LIN {X 89.055,Y 275.987,Z 202.901,A -107.884,B 90.000,C 0.000} C_DIS
LIN {X 91.283,Y 275.258,Z 203.769,A -108.347,B 90.000,C 0.000} C_DIS
LIN {X 93.519,Y 274.506,Z 204.596,A -108.813,B 90.000,C 0.000} C_DIS
LIN {X 95.762,Y 273.732,Z 205.382,A -109.282,B 90.000,C 0.000} C_DIS
LIN {X 98.010,Y 272.935,Z 206.132,A -109.753,B 90.000,C 0.000} C_DIS
LIN {X 100.260,Y 272.116,Z 206.848,A -110.226,B 90.000,C 0.000} C_DIS
LIN {X 102.512,Y 271.277,Z 207.537,A -110.701,B 90.000,C 0.000} C_DIS
LIN {X 104.763,Y 270.415,Z 208.199,A -111.177,B 90.000,C 0.000} C_DIS
LIN {X 107.012,Y 269.533,Z 208.839,A -111.655,B 90.000,C 0.000} C_DIS
LIN {X 109.259,Y 268.630,Z 209.461,A -112.133,B 90.000,C 0.000} C_DIS
LIN {X 111.501,Y 267.707,Z 210.069,A -112.612,B 90.000,C 0.000} C_DIS
LIN {X 113.738,Y 266.764,Z 210.665,A -113.092,B 90.000,C 0.000} C_DIS
LIN {X 115.968,Y 265.800,Z 211.254,A -113.571,B 90.000,C 0.000} C_DIS
LIN {X 118.189,Y 264.816,Z 211.841,A -114.052,B 90.000,C 0.000} C_DIS
LIN {X 120.405,Y 263.818,Z 212.427,A -114.532,B 90.000,C 0.000} C_DIS
LIN {X 122.611,Y 262.801,Z 213.018,A -115.012,B 90.000,C 0.000} C_DIS
LIN {X 124.806,Y 261.767,Z 213.616,A -115.491,B 90.000,C 0.000} C_DIS
LIN {X 126.991,Y 260.715,Z 214.224,A -115.970,B 90.000,C 0.000} C_DIS
LIN {X 129.163,Y 259.646,Z 214.847,A -116.448,B 90.000,C 0.000} C_DIS
LIN {X 131.322,Y 258.561,Z 215.489,A -116.926,B 90.000,C 0.000} C_DIS
LIN {X 133.467,Y 257.462,Z 216.152,A -117.402,B 90.000,C 0.000} C_DIS
LIN {X 135.595,Y 256.346,Z 216.842,A -117.877,B 90.000,C 0.000} C_DIS
LIN {X 137.706,Y 255.218,Z 217.561,A -118.350,B 90.000,C 0.000} C_DIS
LIN {X 139.800,Y 254.078,Z 218.313,A -118.821,B 90.000,C 0.000} C_DIS
LIN {X 141.874,Y 252.926,Z 219.100,A -119.289,B 90.000,C 0.000} C_DIS
LIN {X 143.243,Y 252.153,Z 219.646,A -119.600,B 90.000,C 0.000} C_DIS
LIN {X 142.255,Y 250.414,Z 219.646,A -119.600,B 90.000,C 0.000} C_DIS
WAIT SEC 0.1
RET=EKI_SetBool("oxy","torchState",FALSE)
RET = EKI_Send("oxy","torchState")
LIN {X 133.364,Y 234.764,Z 219.646,A -119.600,B 90.000,C 0.000} C_DIS
LIN {X 126.224,Y 238.679,Z 194.850,A -117.872,B 90.000,C 0.000} C_DIS
LIN {X 134.638,Y 254.591,Z 194.850,A -117.872,B 90.000,C 0.000} C_DIS
LIN {X 135.573,Y 256.359,Z 194.850,A -117.872,B 90.000,C 0.000} C_DIS
WAIT SEC 1.75
RET=EKI_SetBool("oxy","torchState",TRUE)
RET = EKI_Send("oxy","torchState")
LIN {X 137.702,Y 255.221,Z 195.499,A -118.349,B 90.000,C 0.000} C_DIS
LIN {X 139.833,Y 254.060,Z 196.100,A -118.828,B 90.000,C 0.000} C_DIS
LIN {X 141.962,Y 252.876,Z 196.661,A -119.309,B 90.000,C 0.000} C_DIS
LIN {X 144.088,Y 251.672,Z 197.189,A -119.792,B 90.000,C 0.000} C_DIS
LIN {X 146.208,Y 250.445,Z 197.689,A -120.276,B 90.000,C 0.000} C_DIS
LIN {X 148.321,Y 249.199,Z 198.169,A -120.761,B 90.000,C 0.000} C_DIS
LIN {X 150.425,Y 247.933,Z 198.638,A -121.246,B 90.000,C 0.000} C_DIS
LIN {X 152.518,Y 246.648,Z 199.103,A -121.731,B 90.000,C 0.000} C_DIS
LIN {X 154.603,Y 245.350,Z 199.569,A -122.216,B 90.000,C 0.000} C_DIS
LIN {X 156.674,Y 244.034,Z 200.044,A -122.701,B 90.000,C 0.000} C_DIS
LIN {X 158.730,Y 242.701,Z 200.536,A -123.185,B 90.000,C 0.000} C_DIS
LIN {X 159.559,Y 242.159,Z 200.740,A -123.381,B 90.000,C 0.000} C_DIS
LIN {X 158.459,Y 240.488,Z 200.740,A -123.381,B 90.000,C 0.000} C_DIS
WAIT SEC 0.1
RET=EKI_SetBool("oxy","torchState",FALSE)
RET = EKI_Send("oxy","torchState")
LIN {X 148.555,Y 225.458,Z 200.740,A -123.381,B 90.000,C 0.000} C_DIS
LIN {X 166.339,Y 212.677,Z 183.902,A -128.030,B 90.000,C 0.000} C_DIS
LIN {X 177.428,Y 226.855,Z 183.902,A -128.030,B 90.000,C 0.000} C_DIS
LIN {X 178.660,Y 228.430,Z 183.902,A -128.030,B 90.000,C 0.000} C_DIS
WAIT SEC 1.75
RET=EKI_SetBool("oxy","torchState",TRUE)
RET = EKI_Send("oxy","torchState")
LIN {X 180.589,Y 226.908,Z 184.361,A -128.515,B 90.000,C 0.000} C_DIS
LIN {X 182.507,Y 225.367,Z 184.805,A -129.001,B 90.000,C 0.000} C_DIS
LIN {X 184.414,Y 223.810,Z 185.234,A -129.488,B 90.000,C 0.000} C_DIS
LIN {X 186.310,Y 222.234,Z 185.649,A -129.975,B 90.000,C 0.000} C_DIS
LIN {X 188.194,Y 220.640,Z 186.048,A -130.462,B 90.000,C 0.000} C_DIS
LIN {X 190.067,Y 219.029,Z 186.431,A -130.950,B 90.000,C 0.000} C_DIS
LIN {X 191.927,Y 217.401,Z 186.799,A -131.439,B 90.000,C 0.000} C_DIS
LIN {X 193.776,Y 215.755,Z 187.150,A -131.928,B 90.000,C 0.000} C_DIS
LIN {X 195.612,Y 214.092,Z 187.486,A -132.417,B 90.000,C 0.000} C_DIS
LIN {X 197.435,Y 212.412,Z 187.804,A -132.907,B 90.000,C 0.000} C_DIS
LIN {X 199.245,Y 210.715,Z 188.106,A -133.397,B 90.000,C 0.000} C_DIS
LIN {X 201.043,Y 209.002,Z 188.392,A -133.888,B 90.000,C 0.000} C_DIS
LIN {X 202.826,Y 207.271,Z 188.659,A -134.379,B 90.000,C 0.000} C_DIS
LIN {X 204.596,Y 205.524,Z 188.909,A -134.870,B 90.000,C 0.000} C_DIS
LIN {X 206.352,Y 203.760,Z 189.141,A -135.362,B 90.000,C 0.000} C_DIS
LIN {X 208.094,Y 201.980,Z 189.356,A -135.854,B 90.000,C 0.000} C_DIS
LIN {X 209.822,Y 200.184,Z 189.552,A -136.347,B 90.000,C 0.000} C_DIS
LIN {X 211.535,Y 198.372,Z 189.731,A -136.839,B 90.000,C 0.000} C_DIS
LIN {X 213.234,Y 196.545,Z 189.891,A -137.332,B 90.000,C 0.000} C_DIS
LIN {X 214.917,Y 194.703,Z 190.032,A -137.825,B 90.000,C 0.000} C_DIS
LIN {X 216.586,Y 192.846,Z 190.155,A -138.318,B 90.000,C 0.000} C_DIS
LIN {X 218.239,Y 190.973,Z 190.258,A -138.812,B 90.000,C 0.000} C_DIS
LIN {X 219.876,Y 189.087,Z 190.343,A -139.306,B 90.000,C 0.000} C_DIS
LIN {X 221.498,Y 187.185,Z 190.408,A -139.799,B 90.000,C 0.000} C_DIS
LIN {X 223.103,Y 185.270,Z 190.454,A -140.293,B 90.000,C 0.000} C_DIS
LIN {X 224.481,Y 183.598,Z 190.477,A -140.721,B 90.000,C 0.000} C_DIS
LIN {X 222.933,Y 182.331,Z 190.477,A -140.721,B 90.000,C 0.000} C_DIS
WAIT SEC 0.1
RET=EKI_SetBool("oxy","torchState",FALSE)
RET = EKI_Send("oxy","torchState")
LIN {X 209.000,Y 170.936,Z 190.477,A -140.721,B 90.000,C 0.000} C_DIS
LIN {X 223.386,Y 151.653,Z 212.037,A -145.828,B 90.000,C 0.000} C_DIS
LIN {X 238.278,Y 161.763,Z 212.037,A -145.828,B 90.000,C 0.000} C_DIS
LIN {X 239.933,Y 162.887,Z 212.037,A -145.828,B 90.000,C 0.000} C_DIS
WAIT SEC 1.75
RET=EKI_SetBool("oxy","torchState",TRUE)
RET = EKI_Send("oxy","torchState")
LIN {X 238.516,Y 164.946,Z 212.053,A -145.334,B 90.000,C 0.000} C_DIS
LIN {X 237.085,Y 166.995,Z 212.070,A -144.840,B 90.000,C 0.000} C_DIS
LIN {X 235.641,Y 169.035,Z 212.086,A -144.346,B 90.000,C 0.000} C_DIS
LIN {X 234.172,Y 171.058,Z 212.108,A -143.853,B 90.000,C 0.000} C_DIS
LIN {X 232.688,Y 173.069,Z 212.129,A -143.359,B 90.000,C 0.000} C_DIS
LIN {X 231.191,Y 175.071,Z 212.152,A -142.865,B 90.000,C 0.000} C_DIS
LIN {X 229.671,Y 177.055,Z 212.179,A -142.371,B 90.000,C 0.000} C_DIS
LIN {X 228.135,Y 179.028,Z 212.206,A -141.877,B 90.000,C 0.000} C_DIS
LIN {X 226.587,Y 180.990,Z 212.234,A -141.383,B 90.000,C 0.000} C_DIS
LIN {X 225.017,Y 182.935,Z 212.266,A -140.890,B 90.000,C 0.000} C_DIS
LIN {X 223.430,Y 184.866,Z 212.299,A -140.396,B 90.000,C 0.000} C_DIS
LIN {X 221.831,Y 186.787,Z 212.332,A -139.902,B 90.000,C 0.000} C_DIS
LIN {X 220.212,Y 188.691,Z 212.370,A -139.408,B 90.000,C 0.000} C_DIS
LIN {X 218.576,Y 190.581,Z 212.408,A -138.914,B 90.000,C 0.000} C_DIS
LIN {X 216.927,Y 192.459,Z 212.448,A -138.420,B 90.000,C 0.000} C_DIS
LIN {X 215.261,Y 194.322,Z 212.491,A -137.927,B 90.000,C 0.000} C_DIS
LIN {X 213.576,Y 196.168,Z 212.534,A -137.433,B 90.000,C 0.000} C_DIS
LIN {X 211.879,Y 198.003,Z 212.580,A -136.939,B 90.000,C 0.000} C_DIS
LIN {X 210.166,Y 199.822,Z 212.628,A -136.445,B 90.000,C 0.000} C_DIS
LIN {X 208.434,Y 201.624,Z 212.677,A -135.951,B 90.000,C 0.000} C_DIS
LIN {X 206.689,Y 203.414,Z 212.728,A -135.458,B 90.000,C 0.000} C_DIS
LIN {X 204.930,Y 205.189,Z 212.782,A -134.964,B 90.000,C 0.000} C_DIS
LIN {X 203.152,Y 206.945,Z 212.836,A -134.470,B 90.000,C 0.000} C_DIS
LIN {X 201.362,Y 208.688,Z 212.893,A -133.976,B 90.000,C 0.000} C_DIS
LIN {X 199.558,Y 210.418,Z 212.952,A -133.483,B 90.000,C 0.000} C_DIS
LIN {X 197.735,Y 212.127,Z 213.012,A -132.989,B 90.000,C 0.000} C_DIS
LIN {X 195.900,Y 213.824,Z 213.074,A -132.495,B 90.000,C 0.000} C_DIS
LIN {X 194.053,Y 215.506,Z 213.139,A -132.001,B 90.000,C 0.000} C_DIS
LIN {X 192.187,Y 217.169,Z 213.204,A -131.508,B 90.000,C 0.000} C_DIS
LIN {X 191.631,Y 217.664,Z 213.223,A -131.361,B 90.000,C 0.000} C_DIS
LIN {X 190.309,Y 216.163,Z 213.223,A -131.361,B 90.000,C 0.000} C_DIS
WAIT SEC 0.1
RET=EKI_SetBool("oxy","torchState",FALSE)
RET = EKI_Send("oxy","torchState")
LIN {X 178.415,Y 202.653,Z 213.223,A -131.361,B 90.000,C 0.000} C_DIS
LIN {X 175.571,Y 205.122,Z 236.485,A -130.561,B 90.000,C 0.000} C_DIS
LIN {X 187.276,Y 218.796,Z 236.485,A -130.561,B 90.000,C 0.000} C_DIS
LIN {X 188.576,Y 220.316,Z 236.485,A -130.561,B 90.000,C 0.000} C_DIS
WAIT SEC 1.75
RET=EKI_SetBool("oxy","torchState",TRUE)
RET = EKI_Send("oxy","torchState")
LIN {X 190.445,Y 218.694,Z 236.131,A -131.050,B 90.000,C 0.000} C_DIS
LIN {X 192.308,Y 217.065,Z 235.780,A -131.539,B 90.000,C 0.000} C_DIS
LIN {X 194.151,Y 215.411,Z 235.439,A -132.029,B 90.000,C 0.000} C_DIS
LIN {X 195.984,Y 213.745,Z 235.101,A -132.518,B 90.000,C 0.000} C_DIS
LIN {X 197.805,Y 212.065,Z 234.769,A -133.007,B 90.000,C 0.000} C_DIS
LIN {X 199.608,Y 210.363,Z 234.446,A -133.497,B 90.000,C 0.000} C_DIS
LIN {X 201.401,Y 208.652,Z 234.126,A -133.987,B 90.000,C 0.000} C_DIS
LIN {X 203.177,Y 206.921,Z 233.814,A -134.477,B 90.000,C 0.000} C_DIS
LIN {X 204.939,Y 205.174,Z 233.507,A -134.967,B 90.000,C 0.000} C_DIS
LIN {X 206.691,Y 203.417,Z 233.205,A -135.457,B 90.000,C 0.000} C_DIS
LIN {X 208.420,Y 201.636,Z 232.913,A -135.948,B 90.000,C 0.000} C_DIS
LIN {X 210.140,Y 199.845,Z 232.624,A -136.438,B 90.000,C 0.000} C_DIS
LIN {X 211.845,Y 198.039,Z 232.341,A -136.929,B 90.000,C 0.000} C_DIS
LIN {X 213.532,Y 196.215,Z 232.066,A -137.420,B 90.000,C 0.000} C_DIS
LIN {X 215.209,Y 194.381,Z 231.795,A -137.911,B 90.000,C 0.000} C_DIS
LIN {X 216.864,Y 192.527,Z 231.532,A -138.402,B 90.000,C 0.000} C_DIS
LIN {X 218.507,Y 190.660,Z 231.274,A -138.893,B 90.000,C 0.000} C_DIS
LIN {X 220.137,Y 188.782,Z 231.021,A -139.385,B 90.000,C 0.000} C_DIS
LIN {X 221.745,Y 186.883,Z 230.777,A -139.876,B 90.000,C 0.000} C_DIS
LIN {X 223.342,Y 184.976,Z 230.537,A -140.368,B 90.000,C 0.000} C_DIS
LIN {X 224.921,Y 183.052,Z 230.304,A -140.860,B 90.000,C 0.000} C_DIS
LIN {X 226.482,Y 181.113,Z 230.077,A -141.351,B 90.000,C 0.000} C_DIS
LIN {X 228.033,Y 179.165,Z 229.855,A -141.843,B 90.000,C 0.000} C_DIS
LIN {X 229.559,Y 177.197,Z 229.641,A -142.335,B 90.000,C 0.000} C_DIS
LIN {X 231.074,Y 175.219,Z 229.432,A -142.828,B 90.000,C 0.000} C_DIS
LIN {X 232.573,Y 173.229,Z 229.229,A -143.320,B 90.000,C 0.000} C_DIS
LIN {X 234.049,Y 171.222,Z 229.033,A -143.812,B 90.000,C 0.000} C_DIS
LIN {X 235.515,Y 169.206,Z 228.842,A -144.305,B 90.000,C 0.000} C_DIS
LIN {X 236.960,Y 167.174,Z 228.658,A -144.797,B 90.000,C 0.000} C_DIS
LIN {X 238.387,Y 165.130,Z 228.480,A -145.290,B 90.000,C 0.000} C_DIS
LIN {X 239.804,Y 163.077,Z 228.306,A -145.782,B 90.000,C 0.000} C_DIS
LIN {X 241.192,Y 161.005,Z 228.142,A -146.275,B 90.000,C 0.000} C_DIS
LIN {X 242.569,Y 158.925,Z 227.982,A -146.768,B 90.000,C 0.000} C_DIS
LIN {X 243.929,Y 156.834,Z 227.828,A -147.261,B 90.000,C 0.000} C_DIS
LIN {X 245.266,Y 154.727,Z 227.681,A -147.754,B 90.000,C 0.000} C_DIS
LIN {X 246.593,Y 152.613,Z 227.539,A -148.247,B 90.000,C 0.000} C_DIS
LIN {X 247.894,Y 150.483,Z 227.404,A -148.740,B 90.000,C 0.000} C_DIS
LIN {X 249.180,Y 148.343,Z 227.275,A -149.234,B 90.000,C 0.000} C_DIS
LIN {X 250.452,Y 146.195,Z 227.151,A -149.727,B 90.000,C 0.000} C_DIS
LIN {X 251.697,Y 144.030,Z 227.036,A -150.220,B 90.000,C 0.000} C_DIS
LIN {X 252.930,Y 141.859,Z 226.924,A -150.714,B 90.000,C 0.000} C_DIS
LIN {X 254.143,Y 139.675,Z 226.820,A -151.207,B 90.000,C 0.000} C_DIS
LIN {X 255.334,Y 137.480,Z 226.722,A -151.701,B 90.000,C 0.000} C_DIS
LIN {X 256.513,Y 135.278,Z 226.628,A -152.194,B 90.000,C 0.000} C_DIS
LIN {X 257.665,Y 133.061,Z 226.544,A -152.688,B 90.000,C 0.000} C_DIS
LIN {X 258.260,Y 131.917,Z 226.500,A -152.942,B 90.000,C 0.000} C_DIS
LIN {X 256.478,Y 131.007,Z 226.500,A -152.942,B 90.000,C 0.000} C_DIS
WAIT SEC 0.1
RET=EKI_SetBool("oxy","torchState",FALSE)
RET = EKI_Send("oxy","torchState")
LIN {X 240.449,Y 122.819,Z 226.500,A -152.942,B 90.000,C 0.000} C_DIS
LIN {X 242.380,Y 118.962,Z 209.835,A -153.858,B 90.000,C 0.000} C_DIS
LIN {X 258.538,Y 126.893,Z 209.835,A -153.858,B 90.000,C 0.000} C_DIS
LIN {X 260.334,Y 127.774,Z 209.835,A -153.858,B 90.000,C 0.000} C_DIS
WAIT SEC 1.75
RET=EKI_SetBool("oxy","torchState",TRUE)
RET = EKI_Send("oxy","torchState")
LIN {X 261.410,Y 125.557,Z 209.418,A -154.345,B 90.000,C 0.000} C_DIS
LIN {X 262.464,Y 123.338,Z 208.956,A -154.830,B 90.000,C 0.000} C_DIS
LIN {X 263.495,Y 121.118,Z 208.449,A -155.314,B 90.000,C 0.000} C_DIS
LIN {X 264.505,Y 118.898,Z 207.901,A -155.795,B 90.000,C 0.000} C_DIS
LIN {X 265.491,Y 116.679,Z 207.309,A -156.275,B 90.000,C 0.000} C_DIS
LIN {X 266.455,Y 114.460,Z 206.680,A -156.753,B 90.000,C 0.000} C_DIS
LIN {X 267.397,Y 112.243,Z 206.013,A -157.229,B 90.000,C 0.000} C_DIS
LIN {X 268.316,Y 110.027,Z 205.310,A -157.703,B 90.000,C 0.000} C_DIS
LIN {X 269.213,Y 107.813,Z 204.573,A -158.175,B 90.000,C 0.000} C_DIS
LIN {X 270.089,Y 105.601,Z 203.805,A -158.645,B 90.000,C 0.000} C_DIS
LIN {X 270.942,Y 103.392,Z 203.004,A -159.113,B 90.000,C 0.000} C_DIS
LIN {X 271.774,Y 101.185,Z 202.177,A -159.579,B 90.000,C 0.000} C_DIS
LIN {X 272.584,Y 98.981,Z 201.321,A -160.043,B 90.000,C 0.000} C_DIS
LIN {X 273.373,Y 96.779,Z 200.440,A -160.505,B 90.000,C 0.000} C_DIS
LIN {X 274.142,Y 94.579,Z 199.535,A -160.966,B 90.000,C 0.000} C_DIS
LIN {X 274.891,Y 92.381,Z 198.609,A -161.424,B 90.000,C 0.000} C_DIS
LIN {X 275.620,Y 90.186,Z 197.661,A -161.881,B 90.000,C 0.000} C_DIS
LIN {X 276.327,Y 87.993,Z 196.693,A -162.337,B 90.000,C 0.000} C_DIS
LIN {X 277.015,Y 85.801,Z 195.707,A -162.790,B 90.000,C 0.000} C_DIS
LIN {X 277.684,Y 83.610,Z 194.706,A -163.243,B 90.000,C 0.000} C_DIS
LIN {X 278.219,Y 81.819,Z 193.877,A -163.612,B 90.000,C 0.000} C_DIS
LIN {X 276.300,Y 81.255,Z 193.877,A -163.612,B 90.000,C 0.000} C_DIS
WAIT SEC 0.1
RET=EKI_SetBool("oxy","torchState",FALSE)
RET = EKI_Send("oxy","torchState")
LIN {X 259.031,Y 76.177,Z 193.877,A -163.612,B 90.000,C 0.000} C_DIS
LIN {X 263.643,Y 58.244,Z 184.719,A -167.542,B 90.000,C 0.000} C_DIS
LIN {X 281.219,Y 62.127,Z 184.719,A -167.542,B 90.000,C 0.000} C_DIS
LIN {X 283.172,Y 62.558,Z 184.719,A -167.542,B 90.000,C 0.000} C_DIS
WAIT SEC 1.75
RET=EKI_SetBool("oxy","torchState",TRUE)
RET = EKI_Send("oxy","torchState")
LIN {X 283.654,Y 60.332,Z 183.689,A -167.992,B 90.000,C 0.000} C_DIS
LIN {X 284.118,Y 58.098,Z 182.669,A -168.443,B 90.000,C 0.000} C_DIS
LIN {X 284.566,Y 55.856,Z 181.657,A -168.895,B 90.000,C 0.000} C_DIS
LIN {X 284.999,Y 53.608,Z 180.653,A -169.347,B 90.000,C 0.000} C_DIS
LIN {X 285.416,Y 51.354,Z 179.657,A -169.800,B 90.000,C 0.000} C_DIS
LIN {X 285.810,Y 49.091,Z 178.670,A -170.254,B 90.000,C 0.000} C_DIS
LIN {X 286.190,Y 46.824,Z 177.689,A -170.708,B 90.000,C 0.000} C_DIS
LIN {X 286.556,Y 44.552,Z 176.713,A -171.163,B 90.000,C 0.000} C_DIS
LIN {X 286.896,Y 42.272,Z 175.746,A -171.618,B 90.000,C 0.000} C_DIS
LIN {X 287.229,Y 39.990,Z 174.781,A -172.074,B 90.000,C 0.000} C_DIS
LIN {X 287.537,Y 37.702,Z 173.823,A -172.530,B 90.000,C 0.000} C_DIS
LIN {X 287.826,Y 35.409,Z 172.870,A -172.987,B 90.000,C 0.000} C_DIS
LIN {X 288.096,Y 33.113,Z 171.920,A -173.443,B 90.000,C 0.000} C_DIS
LIN {X 288.355,Y 30.814,Z 170.973,A -173.900,B 90.000,C 0.000} C_DIS
LIN {X 288.593,Y 28.512,Z 170.029,A -174.358,B 90.000,C 0.000} C_DIS
LIN {X 288.809,Y 26.206,Z 169.087,A -174.815,B 90.000,C 0.000} C_DIS
LIN {X 289.006,Y 23.898,Z 168.148,A -175.273,B 90.000,C 0.000} C_DIS
LIN {X 289.188,Y 21.589,Z 167.209,A -175.731,B 90.000,C 0.000} C_DIS
LIN {X 289.351,Y 19.277,Z 166.271,A -176.188,B 90.000,C 0.000} C_DIS
LIN {X 289.496,Y 16.965,Z 165.333,A -176.646,B 90.000,C 0.000} C_DIS
LIN {X 289.571,Y 15.760,Z 164.845,A -176.885,B 90.000,C 0.000} C_DIS
LIN {X 287.574,Y 15.651,Z 164.845,A -176.885,B 90.000,C 0.000} C_DIS
WAIT SEC 0.1
RET=EKI_SetBool("oxy","torchState",FALSE)
RET = EKI_Send("oxy","torchState")
LIN {X 269.601,Y 14.673,Z 164.845,A -176.885,B 90.000,C 0.000} C_DIS
LIN {X 269.971,Y -3.924,Z 189.556,A 179.167,B 90.000,C 0.000} C_DIS
LIN {X 287.970,Y -4.186,Z 189.556,A 179.167,B 90.000,C 0.000} C_DIS
LIN {X 289.969,Y -4.215,Z 189.556,A 179.167,B 90.000,C 0.000} C_DIS
WAIT SEC 1.75
RET=EKI_SetBool("oxy","torchState",TRUE)
RET = EKI_Send("oxy","torchState")
LIN {X 289.993,Y -2.041,Z 190.790,A 179.597,B 90.000,C 0.000} C_DIS
LIN {X 290.000,Y 0.164,Z 191.968,A -179.968,B 90.000,C 0.000} C_DIS
LIN {X 289.990,Y 2.393,Z 193.100,A -179.527,B 90.000,C 0.000} C_DIS
LIN {X 289.962,Y 4.639,Z 194.196,A -179.083,B 90.000,C 0.000} C_DIS
LIN {X 289.916,Y 6.896,Z 195.270,A -178.637,B 90.000,C 0.000} C_DIS
LIN {X 289.851,Y 9.157,Z 196.334,A -178.191,B 90.000,C 0.000} C_DIS
LIN {X 289.774,Y 11.418,Z 197.398,A -177.744,B 90.000,C 0.000} C_DIS
LIN {X 289.677,Y 13.673,Z 198.472,A -177.298,B 90.000,C 0.000} C_DIS
LIN {X 289.563,Y 15.915,Z 199.570,A -176.854,B 90.000,C 0.000} C_DIS
LIN {X 289.431,Y 18.139,Z 200.704,A -176.414,B 90.000,C 0.000} C_DIS
LIN {X 289.286,Y 20.339,Z 201.881,A -175.978,B 90.000,C 0.000} C_DIS
LIN {X 289.274,Y 20.512,Z 201.976,A -175.944,B 90.000,C 0.000} C_DIS
LIN {X 287.279,Y 20.371,Z 201.976,A -175.944,B 90.000,C 0.000} C_DIS
WAIT SEC 0.1
RET=EKI_SetBool("oxy","torchState",FALSE)
RET = EKI_Send("oxy","torchState")
LIN {X 269.324,Y 19.097,Z 201.976,A -175.944,B 90.000,C 0.000} C_DIS
LIN {X 268.483,Y 28.585,Z 207.939,A -173.923,B 90.000,C 0.000} C_DIS
LIN {X 286.381,Y 30.491,Z 207.939,A -173.923,B 90.000,C 0.000} C_DIS
LIN {X 288.370,Y 30.703,Z 207.939,A -173.923,B 90.000,C 0.000} C_DIS
WAIT SEC 1.75
RET=EKI_SetBool("oxy","torchState",TRUE)
RET = EKI_Send("oxy","torchState")
LIN {X 288.129,Y 32.886,Z 209.132,A -173.489,B 90.000,C 0.000} C_DIS
LIN {X 287.868,Y 35.095,Z 210.273,A -173.049,B 90.000,C 0.000} C_DIS
LIN {X 287.587,Y 37.328,Z 211.361,A -172.605,B 90.000,C 0.000} C_DIS
LIN {X 287.285,Y 39.582,Z 212.399,A -172.155,B 90.000,C 0.000} C_DIS
LIN {X 286.963,Y 41.856,Z 213.386,A -171.701,B 90.000,C 0.000} C_DIS
LIN {X 286.619,Y 44.147,Z 214.324,A -171.244,B 90.000,C 0.000} C_DIS
LIN {X 286.255,Y 46.454,Z 215.214,A -170.782,B 90.000,C 0.000} C_DIS
LIN {X 285.868,Y 48.776,Z 216.057,A -170.317,B 90.000,C 0.000} C_DIS
LIN {X 285.460,Y 51.110,Z 216.853,A -169.849,B 90.000,C 0.000} C_DIS
LIN {X 285.030,Y 53.455,Z 217.605,A -169.378,B 90.000,C 0.000} C_DIS
LIN {X 284.579,Y 55.808,Z 218.316,A -168.905,B 90.000,C 0.000} C_DIS
LIN {X 284.105,Y 58.171,Z 218.981,A -168.429,B 90.000,C 0.000} C_DIS
LIN {X 283.610,Y 60.540,Z 219.607,A -167.950,B 90.000,C 0.000} C_DIS
LIN {X 283.093,Y 62.914,Z 220.195,A -167.470,B 90.000,C 0.000} C_DIS
LIN {X 282.553,Y 65.292,Z 220.743,A -166.989,B 90.000,C 0.000} C_DIS
LIN {X 281.993,Y 67.674,Z 221.256,A -166.505,B 90.000,C 0.000} C_DIS
LIN {X 281.410,Y 70.057,Z 221.731,A -166.020,B 90.000,C 0.000} C_DIS
LIN {X 280.806,Y 72.442,Z 222.175,A -165.534,B 90.000,C 0.000} C_DIS
LIN {X 280.179,Y 74.827,Z 222.584,A -165.047,B 90.000,C 0.000} C_DIS
LIN {X 279.531,Y 77.212,Z 222.962,A -164.559,B 90.000,C 0.000} C_DIS
LIN {X 278.863,Y 79.595,Z 223.311,A -164.070,B 90.000,C 0.000} C_DIS
LIN {X 278.320,Y 81.473,Z 223.566,A -163.684,B 90.000,C 0.000} C_DIS
LIN {X 276.401,Y 80.911,Z 223.566,A -163.684,B 90.000,C 0.000} C_DIS
WAIT SEC 0.1
RET=EKI_SetBool("oxy","torchState",FALSE)
RET = EKI_Send("oxy","torchState")
LIN {X 259.126,Y 75.854,Z 223.566,A -163.684,B 90.000,C 0.000} C_DIS
LIN {X 257.723,Y 80.490,Z 237.115,A -162.656,B 90.000,C 0.000} C_DIS
LIN {X 274.905,Y 85.856,Z 237.115,A -162.656,B 90.000,C 0.000} C_DIS
LIN {X 276.814,Y 86.452,Z 237.115,A -162.656,B 90.000,C 0.000} C_DIS
WAIT SEC 1.75
RET=EKI_SetBool("oxy","torchState",TRUE)
RET = EKI_Send("oxy","torchState")
LIN {X 277.546,Y 84.069,Z 237.291,A -163.148,B 90.000,C 0.000} C_DIS
LIN {X 278.260,Y 81.678,Z 237.445,A -163.641,B 90.000,C 0.000} C_DIS
LIN {X 278.952,Y 79.280,Z 237.571,A -164.135,B 90.000,C 0.000} C_DIS
LIN {X 279.624,Y 76.874,Z 237.673,A -164.628,B 90.000,C 0.000} C_DIS
LIN {X 280.276,Y 74.462,Z 237.751,A -165.122,B 90.000,C 0.000} C_DIS
LIN {X 280.909,Y 72.044,Z 237.804,A -165.615,B 90.000,C 0.000} C_DIS
LIN {X 281.518,Y 69.620,Z 237.829,A -166.109,B 90.000,C 0.000} C_DIS
LIN {X 282.107,Y 67.191,Z 237.830,A -166.603,B 90.000,C 0.000} C_DIS
LIN {X 282.676,Y 64.757,Z 237.807,A -167.097,B 90.000,C 0.000} C_DIS
LIN {X 283.225,Y 62.319,Z 237.759,A -167.591,B 90.000,C 0.000} C_DIS
LIN {X 283.750,Y 59.876,Z 237.684,A -168.084,B 90.000,C 0.000} C_DIS
LIN {X 284.255,Y 57.430,Z 237.585,A -168.578,B 90.000,C 0.000} C_DIS
LIN {X 284.739,Y 54.981,Z 237.461,A -169.071,B 90.000,C 0.000} C_DIS
LIN {X 285.203,Y 52.529,Z 237.313,A -169.564,B 90.000,C 0.000} C_DIS
LIN {X 285.643,Y 50.074,Z 237.138,A -170.057,B 90.000,C 0.000} C_DIS
LIN {X 286.062,Y 47.618,Z 236.939,A -170.549,B 90.000,C 0.000} C_DIS
LIN {X 286.461,Y 45.160,Z 236.715,A -171.041,B 90.000,C 0.000} C_DIS
LIN {X 286.532,Y 44.715,Z 236.673,A -171.130,B 90.000,C 0.000} C_DIS
LIN {X 284.556,Y 44.406,Z 236.673,A -171.130,B 90.000,C 0.000} C_DIS
WAIT SEC 0.1
RET=EKI_SetBool("oxy","torchState",FALSE)
RET = EKI_Send("oxy","torchState")
LIN {X 266.771,Y 41.631,Z 236.673,A -171.130,B 90.000,C 0.000} C_DIS
LIN {X 269.988,Y 2.525,Z 228.878,A -179.464,B 90.000,C 0.000} C_DIS
LIN {X 287.987,Y 2.694,Z 228.878,A -179.464,B 90.000,C 0.000} C_DIS
LIN {X 289.987,Y 2.712,Z 228.878,A -179.464,B 90.000,C 0.000} C_DIS
WAIT SEC 1.75
RET=EKI_SetBool("oxy","torchState",TRUE)
RET = EKI_Send("oxy","torchState")
LIN {X 289.999,Y 0.306,Z 228.200,A -179.939,B 90.000,C 0.000} C_DIS
LIN {X 289.991,Y -2.093,Z 227.499,A 179.586,B 90.000,C 0.000} C_DIS
LIN {X 289.964,Y -4.486,Z 226.775,A 179.114,B 90.000,C 0.000} C_DIS
LIN {X 289.917,Y -6.871,Z 226.031,A 178.642,B 90.000,C 0.000} C_DIS
LIN {X 289.851,Y -9.251,Z 225.267,A 178.172,B 90.000,C 0.000} C_DIS
LIN {X 289.766,Y -11.623,Z 224.484,A 177.703,B 90.000,C 0.000} C_DIS
LIN {X 289.662,Y -13.988,Z 223.682,A 177.235,B 90.000,C 0.000} C_DIS
LIN {X 289.539,Y -16.346,Z 222.862,A 176.769,B 90.000,C 0.000} C_DIS
LIN {X 289.397,Y -18.698,Z 222.026,A 176.303,B 90.000,C 0.000} C_DIS
LIN {X 289.236,Y -21.042,Z 221.174,A 175.839,B 90.000,C 0.000} C_DIS
LIN {X 289.056,Y -23.380,Z 220.307,A 175.376,B 90.000,C 0.000} C_DIS
LIN {X 288.857,Y -25.711,Z 219.426,A 174.914,B 90.000,C 0.000} C_DIS
LIN {X 288.640,Y -28.035,Z 218.532,A 174.452,B 90.000,C 0.000} C_DIS
LIN {X 288.404,Y -30.353,Z 217.626,A 173.992,B 90.000,C 0.000} C_DIS
LIN {X 288.151,Y -32.664,Z 216.709,A 173.533,B 90.000,C 0.000} C_DIS
LIN {X 287.971,Y -34.248,Z 216.077,A 173.218,B 90.000,C 0.000} C_DIS
LIN {X 285.985,Y -34.011,Z 216.077,A 173.218,B 90.000,C 0.000} C_DIS
WAIT SEC 0.1
RET=EKI_SetBool("oxy","torchState",FALSE)
RET = EKI_Send("oxy","torchState")
LIN {X 268.111,Y -31.886,Z 216.077,A 173.218,B 90.000,C 0.000} C_DIS
LIN {X 267.638,Y -35.633,Z 232.790,A 172.416,B 90.000,C 0.000} C_DIS
LIN {X 285.481,Y -38.008,Z 232.790,A 172.416,B 90.000,C 0.000} C_DIS
LIN {X 287.463,Y -38.272,Z 232.790,A 172.416,B 90.000,C 0.000} C_DIS
WAIT SEC 1.75
RET=EKI_SetBool("oxy","torchState",TRUE)
RET = EKI_Send("oxy","torchState")
LIN {X 287.172,Y -40.399,Z 231.509,A 171.992,B 90.000,C 0.000} C_DIS
LIN {X 286.855,Y -42.592,Z 230.352,A 171.555,B 90.000,C 0.000} C_DIS
LIN {X 286.512,Y -44.843,Z 229.320,A 171.105,B 90.000,C 0.000} C_DIS
LIN {X 286.142,Y -47.142,Z 228.412,A 170.644,B 90.000,C 0.000} C_DIS
LIN {X 285.747,Y -49.482,Z 227.626,A 170.176,B 90.000,C 0.000} C_DIS
LIN {X 285.326,Y -51.854,Z 226.959,A 169.700,B 90.000,C 0.000} C_DIS
LIN {X 284.880,Y -54.251,Z 226.408,A 169.218,B 90.000,C 0.000} C_DIS
LIN {X 284.409,Y -56.667,Z 225.972,A 168.732,B 90.000,C 0.000} C_DIS
LIN {X 283.915,Y -59.096,Z 225.650,A 168.242,B 90.000,C 0.000} C_DIS
LIN {X 283.397,Y -61.532,Z 225.435,A 167.750,B 90.000,C 0.000} C_DIS
LIN {X 282.856,Y -63.970,Z 225.331,A 167.256,B 90.000,C 0.000} C_DIS
LIN {X 282.558,Y -65.277,Z 225.316,A 166.992,B 90.000,C 0.000} C_DIS
LIN {X 280.609,Y -64.826,Z 225.316,A 166.992,B 90.000,C 0.000} C_DIS
WAIT SEC 0.1
RET=EKI_SetBool("oxy","torchState",FALSE)
RET = EKI_Send("oxy","torchState")
LIN {X 263.071,Y -60.775,Z 225.316,A 166.992,B 90.000,C 0.000} C_DIS
LIN {X 262.698,Y -62.368,Z 205.443,A 166.644,B 90.000,C 0.000} C_DIS
LIN {X 280.211,Y -66.526,Z 205.443,A 166.644,B 90.000,C 0.000} C_DIS
LIN {X 282.157,Y -66.988,Z 205.443,A 166.644,B 90.000,C 0.000} C_DIS
WAIT SEC 1.75
RET=EKI_SetBool("oxy","torchState",TRUE)
RET = EKI_Send("oxy","torchState")
LIN {X 281.573,Y -69.401,Z 205.149,A 166.154,B 90.000,C 0.000} C_DIS
LIN {X 280.967,Y -71.817,Z 204.946,A 165.662,B 90.000,C 0.000} C_DIS
LIN {X 280.337,Y -74.234,Z 204.837,A 165.168,B 90.000,C 0.000} C_DIS
LIN {X 279.687,Y -76.648,Z 204.817,A 164.674,B 90.000,C 0.000} C_DIS
LIN {X 279.017,Y -79.055,Z 204.882,A 164.181,B 90.000,C 0.000} C_DIS
LIN {X 278.326,Y -81.453,Z 205.033,A 163.688,B 90.000,C 0.000} C_DIS
LIN {X 277.616,Y -83.838,Z 205.264,A 163.196,B 90.000,C 0.000} C_DIS
LIN {X 276.889,Y -86.210,Z 205.571,A 162.706,B 90.000,C 0.000} C_DIS
LIN {X 276.144,Y -88.566,Z 205.951,A 162.218,B 90.000,C 0.000} C_DIS
LIN {X 275.384,Y -90.904,Z 206.402,A 161.732,B 90.000,C 0.000} C_DIS
LIN {X 274.607,Y -93.223,Z 206.920,A 161.249,B 90.000,C 0.000} C_DIS
LIN {X 273.816,Y -95.521,Z 207.503,A 160.769,B 90.000,C 0.000} C_DIS
LIN {X 273.011,Y -97.798,Z 208.147,A 160.291,B 90.000,C 0.000} C_DIS
LIN {X 272.193,Y -100.053,Z 208.850,A 159.817,B 90.000,C 0.000} C_DIS
LIN {X 271.362,Y -102.286,Z 209.609,A 159.347,B 90.000,C 0.000} C_DIS
LIN {X 270.519,Y -104.494,Z 210.420,A 158.880,B 90.000,C 0.000} C_DIS
LIN {X 269.665,Y -106.680,Z 211.282,A 158.416,B 90.000,C 0.000} C_DIS
LIN {X 268.800,Y -108.842,Z 212.192,A 157.956,B 90.000,C 0.000} C_DIS
LIN {X 268.290,Y -110.093,Z 212.745,A 157.689,B 90.000,C 0.000} C_DIS
LIN {X 266.440,Y -109.334,Z 212.745,A 157.689,B 90.000,C 0.000} C_DIS
WAIT SEC 0.1
RET=EKI_SetBool("oxy","torchState",FALSE)
RET = EKI_Send("oxy","torchState")
LIN {X 249.787,Y -102.501,Z 212.745,A 157.689,B 90.000,C 0.000} C_DIS
LIN {X 254.981,Y -88.797,Z 231.272,A 160.799,B 90.000,C 0.000} C_DIS
LIN {X 271.979,Y -94.717,Z 231.272,A 160.799,B 90.000,C 0.000} C_DIS
LIN {X 273.868,Y -95.375,Z 231.272,A 160.799,B 90.000,C 0.000} C_DIS
WAIT SEC 1.75
RET=EKI_SetBool("oxy","torchState",TRUE)
RET = EKI_Send("oxy","torchState")
LIN {X 273.073,Y -97.625,Z 232.015,A 160.328,B 90.000,C 0.000} C_DIS
LIN {X 272.258,Y -99.865,Z 232.767,A 159.857,B 90.000,C 0.000} C_DIS
LIN {X 271.428,Y -102.101,Z 233.518,A 159.386,B 90.000,C 0.000} C_DIS
LIN {X 270.582,Y -104.331,Z 234.266,A 158.914,B 90.000,C 0.000} C_DIS
LIN {X 269.714,Y -106.556,Z 235.001,A 158.442,B 90.000,C 0.000} C_DIS
LIN {X 268.825,Y -108.780,Z 235.719,A 157.969,B 90.000,C 0.000} C_DIS
LIN {X 267.915,Y -111.002,Z 236.412,A 157.495,B 90.000,C 0.000} C_DIS
LIN {X 266.982,Y -113.225,Z 237.072,A 157.018,B 90.000,C 0.000} C_DIS
LIN {X 266.028,Y -115.450,Z 237.698,A 156.540,B 90.000,C 0.000} C_DIS
LIN {X 265.051,Y -117.676,Z 238.277,A 156.060,B 90.000,C 0.000} C_DIS
LIN {X 264.050,Y -119.905,Z 238.804,A 155.577,B 90.000,C 0.000} C_DIS
LIN {X 263.025,Y -122.137,Z 239.274,A 155.092,B 90.000,C 0.000} C_DIS
LIN {X 262.177,Y -123.949,Z 239.609,A 154.697,B 90.000,C 0.000} C_DIS
LIN {X 260.369,Y -123.094,Z 239.609,A 154.697,B 90.000,C 0.000} C_DIS
WAIT SEC 0.1
RET=EKI_SetBool("oxy","torchState",FALSE)
RET = EKI_Send("oxy","torchState")
LIN {X 244.096,Y -115.400,Z 239.609,A 154.697,B 90.000,C 0.000} C_DIS
LIN {X 241.168,Y -121.400,Z 222.499,A 153.280,B 90.000,C 0.000} C_DIS
LIN {X 257.246,Y -129.494,Z 222.499,A 153.280,B 90.000,C 0.000} C_DIS
LIN {X 259.032,Y -130.393,Z 222.499,A 153.280,B 90.000,C 0.000} C_DIS
WAIT SEC 1.75
RET=EKI_SetBool("oxy","torchState",TRUE)
RET = EKI_Send("oxy","torchState")
LIN {X 257.965,Y -132.492,Z 223.338,A 152.815,B 90.000,C 0.000} C_DIS
LIN {X 256.870,Y -134.602,Z 224.109,A 152.345,B 90.000,C 0.000} C_DIS
LIN {X 255.748,Y -136.722,Z 224.813,A 151.871,B 90.000,C 0.000} C_DIS
LIN {X 254.599,Y -138.849,Z 225.451,A 151.394,B 90.000,C 0.000} C_DIS
LIN {X 253.425,Y -140.981,Z 226.020,A 150.913,B 90.000,C 0.000} C_DIS
LIN {X 252.225,Y -143.116,Z 226.521,A 150.429,B 90.000,C 0.000} C_DIS
LIN {X 251.001,Y -145.252,Z 226.952,A 149.942,B 90.000,C 0.000} C_DIS
LIN {X 249.753,Y -147.388,Z 227.314,A 149.454,B 90.000,C 0.000} C_DIS
LIN {X 248.482,Y -149.520,Z 227.606,A 148.963,B 90.000,C 0.000} C_DIS
LIN {X 247.189,Y -151.649,Z 227.827,A 148.471,B 90.000,C 0.000} C_DIS
LIN {X 245.875,Y -153.770,Z 227.974,A 147.978,B 90.000,C 0.000} C_DIS
LIN {X 244.541,Y -155.882,Z 228.047,A 147.485,B 90.000,C 0.000} C_DIS
LIN {X 244.051,Y -156.649,Z 228.058,A 147.305,B 90.000,C 0.000} C_DIS
LIN {X 242.368,Y -155.569,Z 228.058,A 147.305,B 90.000,C 0.000} C_DIS
WAIT SEC 0.1
RET=EKI_SetBool("oxy","torchState",FALSE)
RET = EKI_Send("oxy","torchState")
LIN {X 227.220,Y -145.846,Z 228.058,A 147.305,B 90.000,C 0.000} C_DIS
LIN {X 225.096,Y -149.103,Z 205.774,A 146.480,B 90.000,C 0.000} C_DIS
LIN {X 240.103,Y -159.043,Z 205.774,A 146.480,B 90.000,C 0.000} C_DIS
LIN {X 241.770,Y -160.147,Z 205.774,A 146.480,B 90.000,C 0.000} C_DIS
WAIT SEC 1.75
RET=EKI_SetBool("oxy","torchState",TRUE)
RET = EKI_Send("oxy","torchState")
LIN {X 243.128,Y -158.077,Z 206.118,A 146.969,B 90.000,C 0.000} C_DIS
LIN {X 244.474,Y -155.987,Z 206.381,A 147.460,B 90.000,C 0.000} C_DIS
LIN {X 245.807,Y -153.880,Z 206.560,A 147.953,B 90.000,C 0.000} C_DIS
LIN {X 247.123,Y -151.756,Z 206.647,A 148.446,B 90.000,C 0.000} C_DIS
LIN {X 248.422,Y -149.621,Z 206.638,A 148.940,B 90.000,C 0.000} C_DIS
LIN {X 249.701,Y -147.476,Z 206.529,A 149.433,B 90.000,C 0.000} C_DIS
LIN {X 250.959,Y -145.326,Z 206.314,A 149.926,B 90.000,C 0.000} C_DIS
LIN {X 252.191,Y -143.176,Z 205.987,A 150.415,B 90.000,C 0.000} C_DIS
LIN {X 253.397,Y -141.032,Z 205.544,A 150.901,B 90.000,C 0.000} C_DIS
LIN {X 254.572,Y -138.899,Z 204.981,A 151.382,B 90.000,C 0.000} C_DIS
LIN {X 255.714,Y -136.785,Z 204.291,A 151.857,B 90.000,C 0.000} C_DIS
LIN {X 255.789,Y -136.646,Z 204.242,A 151.888,B 90.000,C 0.000} C_DIS
LIN {X 254.025,Y -135.704,Z 204.242,A 151.888,B 90.000,C 0.000} C_DIS
WAIT SEC 0.1
RET=EKI_SetBool("oxy","torchState",FALSE)
RET = EKI_Send("oxy","torchState")
LIN {X 238.148,Y -127.222,Z 204.242,A 151.888,B 90.000,C 0.000} C_DIS
LIN {X 246.938,Y -109.187,Z 187.871,A 156.147,B 90.000,C 0.000} C_DIS
LIN {X 263.400,Y -116.466,Z 187.871,A 156.147,B 90.000,C 0.000} C_DIS
LIN {X 265.229,Y -117.275,Z 187.871,A 156.147,B 90.000,C 0.000} C_DIS
WAIT SEC 1.75
RET=EKI_SetBool("oxy","torchState",TRUE)
RET = EKI_Send("oxy","torchState")
LIN {X 265.712,Y -116.177,Z 185.678,A 156.384,B 90.000,C 0.000} C_DIS
LIN {X 266.132,Y -115.212,Z 183.411,A 156.592,B 90.000,C 0.000} C_DIS
LIN {X 266.499,Y -114.360,Z 181.090,A 156.775,B 90.000,C 0.000} C_DIS
LIN {X 266.824,Y -113.601,Z 178.730,A 156.938,B 90.000,C 0.000} C_DIS
LIN {X 267.117,Y -112.910,Z 176.346,A 157.086,B 90.000,C 0.000} C_DIS
LIN {X 267.389,Y -112.264,Z 173.947,A 157.225,B 90.000,C 0.000} C_DIS
LIN {X 267.651,Y -111.636,Z 171.541,A 157.359,B 90.000,C 0.000} C_DIS
LIN {X 267.914,Y -111.006,Z 169.137,A 157.494,B 90.000,C 0.000} C_DIS
LIN {X 268.186,Y -110.346,Z 166.741,A 157.635,B 90.000,C 0.000} C_DIS
LIN {X 268.293,Y -110.086,Z 165.841,A 157.691,B 90.000,C 0.000} C_DIS
LIN {X 266.443,Y -109.326,Z 165.841,A 157.691,B 90.000,C 0.000} C_DIS
WAIT SEC 0.1
RET=EKI_SetBool("oxy","torchState",FALSE)
RET = EKI_Send("oxy","torchState")
LIN {X 249.790,Y -102.493,Z 165.841,A 157.691,B 90.000,C 0.000} C_DIS
LIN {X 251.429,Y -98.404,Z 155.153,A 158.626,B 90.000,C 0.000} C_DIS
LIN {X 268.191,Y -104.965,Z 155.153,A 158.626,B 90.000,C 0.000} C_DIS
LIN {X 270.053,Y -105.694,Z 155.153,A 158.626,B 90.000,C 0.000} C_DIS
WAIT SEC 1.75
RET=EKI_SetBool("oxy","torchState",TRUE)
RET = EKI_Send("oxy","torchState")
LIN {X 270.572,Y -104.359,Z 153.103,A 158.908,B 90.000,C 0.000} C_DIS
LIN {X 271.148,Y -102.853,Z 151.194,A 159.227,B 90.000,C 0.000} C_DIS
LIN {X 271.781,Y -101.169,Z 149.459,A 159.583,B 90.000,C 0.000} C_DIS
LIN {X 272.467,Y -99.306,Z 147.939,A 159.975,B 90.000,C 0.000} C_DIS
LIN {X 273.200,Y -97.271,Z 146.686,A 160.402,B 90.000,C 0.000} C_DIS
LIN {X 273.966,Y -95.094,Z 145.726,A 160.858,B 90.000,C 0.000} C_DIS
LIN {X 274.747,Y -92.813,Z 145.066,A 161.334,B 90.000,C 0.000} C_DIS
LIN {X 275.528,Y -90.468,Z 144.694,A 161.823,B 90.000,C 0.000} C_DIS
LIN {X 276.297,Y -88.091,Z 144.600,A 162.316,B 90.000,C 0.000} C_DIS
LIN {X 276.701,Y -86.815,Z 144.660,A 162.581,B 90.000,C 0.000} C_DIS
LIN {X 274.792,Y -86.216,Z 144.660,A 162.581,B 90.000,C 0.000} C_DIS
WAIT SEC 0.1
RET=EKI_SetBool("oxy","torchState",FALSE)
RET = EKI_Send("oxy","torchState")
LIN {X 257.618,Y -80.827,Z 144.660,A 162.581,B 90.000,C 0.000} C_DIS
LIN {X 262.894,Y -61.535,Z 153.240,A 166.826,B 90.000,C 0.000} C_DIS
LIN {X 280.421,Y -65.637,Z 153.240,A 166.826,B 90.000,C 0.000} C_DIS
LIN {X 282.368,Y -66.093,Z 153.240,A 166.826,B 90.000,C 0.000} C_DIS
WAIT SEC 1.75
RET=EKI_SetBool("oxy","torchState",TRUE)
RET = EKI_Send("oxy","torchState")
LIN {X 282.860,Y -63.951,Z 154.432,A 167.260,B 90.000,C 0.000} C_DIS
LIN {X 283.338,Y -61.795,Z 155.602,A 167.697,B 90.000,C 0.000} C_DIS
LIN {X 283.803,Y -59.625,Z 156.753,A 168.135,B 90.000,C 0.000} C_DIS
LIN {X 284.253,Y -57.444,Z 157.888,A 168.575,B 90.000,C 0.000} C_DIS
LIN {X 284.686,Y -55.253,Z 159.011,A 169.016,B 90.000,C 0.000} C_DIS
LIN {X 285.101,Y -53.054,Z 160.126,A 169.458,B 90.000,C 0.000} C_DIS
LIN {X 285.503,Y -50.852,Z 161.237,A 169.901,B 90.000,C 0.000} C_DIS
LIN {X 285.887,Y -48.645,Z 162.347,A 170.343,B 90.000,C 0.000} C_DIS
LIN {X 286.256,Y -46.437,Z 163.459,A 170.786,B 90.000,C 0.000} C_DIS
LIN {X 286.607,Y -44.229,Z 164.578,A 171.227,B 90.000,C 0.000} C_DIS
LIN {X 286.939,Y -42.024,Z 165.708,A 171.668,B 90.000,C 0.000} C_DIS
LIN {X 287.253,Y -39.824,Z 166.851,A 172.107,B 90.000,C 0.000} C_DIS
LIN {X 287.548,Y -37.630,Z 168.013,A 172.544,B 90.000,C 0.000} C_DIS
LIN {X 287.825,Y -35.446,Z 169.197,A 172.979,B 90.000,C 0.000} C_DIS
LIN {X 288.084,Y -33.273,Z 170.405,A 173.412,B 90.000,C 0.000} C_DIS
LIN {X 288.326,Y -31.114,Z 171.641,A 173.841,B 90.000,C 0.000} C_DIS
LIN {X 288.548,Y -28.972,Z 172.911,A 174.266,B 90.000,C 0.000} C_DIS
LIN {X 288.754,Y -26.849,Z 174.215,A 174.688,B 90.000,C 0.000} C_DIS
LIN {X 288.942,Y -24.749,Z 175.556,A 175.104,B 90.000,C 0.000} C_DIS
LIN {X 288.994,Y -24.137,Z 175.958,A 175.226,B 90.000,C 0.000} C_DIS
LIN {X 287.001,Y -23.971,Z 175.958,A 175.226,B 90.000,C 0.000} C_DIS
WAIT SEC 0.1
RET=EKI_SetBool("oxy","torchState",FALSE)
RET = EKI_Send("oxy","torchState")
LIN {X 269.063,Y -22.473,Z 175.958,A 175.226,B 90.000,C 0.000} C_DIS
LIN {X 269.271,Y -19.828,Z 148.713,A 175.789,B 90.000,C 0.000} C_DIS
LIN {X 287.222,Y -21.150,Z 148.713,A 175.789,B 90.000,C 0.000} C_DIS
LIN {X 289.217,Y -21.297,Z 148.713,A 175.789,B 90.000,C 0.000} C_DIS
WAIT SEC 1.75
RET=EKI_SetBool("oxy","torchState",TRUE)
RET = EKI_Send("oxy","torchState")
LIN {X 289.042,Y -23.524,Z 147.592,A 175.347,B 90.000,C 0.000} C_DIS
LIN {X 288.855,Y -25.744,Z 146.458,A 174.907,B 90.000,C 0.000} C_DIS
LIN {X 288.649,Y -27.954,Z 145.309,A 174.468,B 90.000,C 0.000} C_DIS
LIN {X 288.427,Y -30.157,Z 144.148,A 174.031,B 90.000,C 0.000} C_DIS
LIN {X 288.186,Y -32.354,Z 142.980,A 173.594,B 90.000,C 0.000} C_DIS
LIN {X 287.931,Y -34.547,Z 141.808,A 173.158,B 90.000,C 0.000} C_DIS
LIN {X 287.656,Y -36.737,Z 140.634,A 172.722,B 90.000,C 0.000} C_DIS
LIN {X 287.373,Y -38.926,Z 139.461,A 172.286,B 90.000,C 0.000} C_DIS
LIN {X 287.070,Y -41.114,Z 138.292,A 171.849,B 90.000,C 0.000} C_DIS
LIN {X 286.747,Y -43.305,Z 137.131,A 171.412,B 90.000,C 0.000} C_DIS
LIN {X 286.407,Y -45.498,Z 135.980,A 170.974,B 90.000,C 0.000} C_DIS
LIN {X 286.050,Y -47.695,Z 134.843,A 170.534,B 90.000,C 0.000} C_DIS
LIN {X 285.675,Y -49.897,Z 133.721,A 170.092,B 90.000,C 0.000} C_DIS
LIN {X 285.279,Y -52.107,Z 132.622,A 169.649,B 90.000,C 0.000} C_DIS
LIN {X 284.865,Y -54.324,Z 131.544,A 169.203,B 90.000,C 0.000} C_DIS
LIN {X 284.433,Y -56.549,Z 130.491,A 168.755,B 90.000,C 0.000} C_DIS
LIN {X 284.132,Y -58.041,Z 129.805,A 168.455,B 90.000,C 0.000} C_DIS
LIN {X 282.173,Y -57.641,Z 129.805,A 168.455,B 90.000,C 0.000} C_DIS
WAIT SEC 0.1
RET=EKI_SetBool("oxy","torchState",FALSE)
RET = EKI_Send("oxy","torchState")
LIN {X 264.537,Y -54.038,Z 129.805,A 168.455,B 90.000,C 0.000} C_DIS
LIN {X 267.894,Y -33.660,Z 110.915,A 172.838,B 90.000,C 0.000} C_DIS
LIN {X 285.753,Y -35.904,Z 110.915,A 172.838,B 90.000,C 0.000} C_DIS
LIN {X 287.738,Y -36.153,Z 110.915,A 172.838,B 90.000,C 0.000} C_DIS
WAIT SEC 1.75
RET=EKI_SetBool("oxy","torchState",TRUE)
RET = EKI_Send("oxy","torchState")
LIN {X 288.010,Y -33.880,Z 111.919,A 173.291,B 90.000,C 0.000} C_DIS
LIN {X 288.269,Y -31.607,Z 112.924,A 173.743,B 90.000,C 0.000} C_DIS
LIN {X 288.510,Y -29.332,Z 113.933,A 174.195,B 90.000,C 0.000} C_DIS
LIN {X 288.735,Y -27.058,Z 114.947,A 174.646,B 90.000,C 0.000} C_DIS
LIN {X 288.938,Y -24.786,Z 115.970,A 175.097,B 90.000,C 0.000} C_DIS
LIN {X 289.124,Y -22.518,Z 117.002,A 175.547,B 90.000,C 0.000} C_DIS
LIN {X 289.292,Y -20.253,Z 118.046,A 175.995,B 90.000,C 0.000} C_DIS
LIN {X 289.441,Y -17.993,Z 119.105,A 176.443,B 90.000,C 0.000} C_DIS
LIN {X 289.572,Y -15.740,Z 120.180,A 176.889,B 90.000,C 0.000} C_DIS
LIN {X 289.685,Y -13.495,Z 121.274,A 177.333,B 90.000,C 0.000} C_DIS
LIN {X 289.780,Y -11.260,Z 122.388,A 177.775,B 90.000,C 0.000} C_DIS
LIN {X 289.858,Y -9.035,Z 123.524,A 178.215,B 90.000,C 0.000} C_DIS
LIN {X 289.920,Y -6.821,Z 124.683,A 178.652,B 90.000,C 0.000} C_DIS
LIN {X 289.963,Y -4.621,Z 125.870,A 179.087,B 90.000,C 0.000} C_DIS
LIN {X 289.989,Y -2.436,Z 127.083,A 179.519,B 90.000,C 0.000} C_DIS
LIN {X 289.998,Y -0.262,Z 128.317,A 179.948,B 90.000,C 0.000} C_DIS
LIN {X 289.992,Y 1.908,Z 129.559,A -179.623,B 90.000,C 0.000} C_DIS
LIN {X 289.971,Y 4.076,Z 130.802,A -179.195,B 90.000,C 0.000} C_DIS
LIN {X 289.932,Y 6.251,Z 132.034,A -178.765,B 90.000,C 0.000} C_DIS
LIN {X 289.903,Y 7.516,Z 132.741,A -178.515,B 90.000,C 0.000} C_DIS
LIN {X 287.903,Y 7.464,Z 132.741,A -178.515,B 90.000,C 0.000} C_DIS
WAIT SEC 0.1
RET=EKI_SetBool("oxy","torchState",FALSE)
RET = EKI_Send("oxy","torchState")
LIN {X 269.909,Y 6.998,Z 132.741,A -178.515,B 90.000,C 0.000} C_DIS
LIN {X 267.363,Y 37.645,Z 110.248,A -171.985,B 90.000,C 0.000} C_DIS
LIN {X 285.187,Y 40.155,Z 110.248,A -171.985,B 90.000,C 0.000} C_DIS
LIN {X 287.167,Y 40.434,Z 110.248,A -171.985,B 90.000,C 0.000} C_DIS
WAIT SEC 1.75
RET=EKI_SetBool("oxy","torchState",TRUE)
RET = EKI_Send("oxy","torchState")
LIN {X 287.482,Y 38.121,Z 109.354,A -172.446,B 90.000,C 0.000} C_DIS
LIN {X 287.776,Y 35.808,Z 108.454,A -172.907,B 90.000,C 0.000} C_DIS
LIN {X 288.054,Y 33.494,Z 107.548,A -173.368,B 90.000,C 0.000} C_DIS
LIN {X 288.318,Y 31.181,Z 106.638,A -173.828,B 90.000,C 0.000} C_DIS
LIN {X 288.554,Y 28.868,Z 105.719,A -174.287,B 90.000,C 0.000} C_DIS
LIN {X 288.777,Y 26.556,Z 104.797,A -174.746,B 90.000,C 0.000} C_DIS
LIN {X 288.982,Y 24.244,Z 103.868,A -175.204,B 90.000,C 0.000} C_DIS
LIN {X 289.164,Y 21.933,Z 102.932,A -175.662,B 90.000,C 0.000} C_DIS
LIN {X 289.333,Y 19.623,Z 101.992,A -176.120,B 90.000,C 0.000} C_DIS
LIN {X 289.479,Y 17.315,Z 101.045,A -176.577,B 90.000,C 0.000} C_DIS
LIN {X 289.606,Y 15.007,Z 100.092,A -177.034,B 90.000,C 0.000} C_DIS
LIN {X 289.721,Y 12.701,Z 99.135,A -177.490,B 90.000,C 0.000} C_DIS
LIN {X 289.808,Y 10.397,Z 98.169,A -177.945,B 90.000,C 0.000} C_DIS
LIN {X 289.882,Y 8.094,Z 97.199,A -178.401,B 90.000,C 0.000} C_DIS
LIN {X 289.941,Y 5.793,Z 96.224,A -178.855,B 90.000,C 0.000} C_DIS
LIN {X 289.973,Y 3.496,Z 95.241,A -179.309,B 90.000,C 0.000} C_DIS
LIN {X 289.994,Y 1.199,Z 94.254,A -179.763,B 90.000,C 0.000} C_DIS
LIN {X 289.995,Y -1.095,Z 93.260,A 179.784,B 90.000,C 0.000} C_DIS
LIN {X 289.995,Y -1.751,Z 92.975,A 179.654,B 90.000,C 0.000} C_DIS
LIN {X 287.995,Y -1.739,Z 92.975,A 179.654,B 90.000,C 0.000} C_DIS
WAIT SEC 0.1
RET=EKI_SetBool("oxy","torchState",FALSE)
RET = EKI_Send("oxy","torchState")
LIN {X 269.995,Y -1.630,Z 92.975,A 179.654,B 90.000,C 0.000} C_DIS
LIN {X 266.781,Y -41.566,Z 74.133,A 171.144,B 90.000,C 0.000} C_DIS
LIN {X 284.567,Y -44.337,Z 74.133,A 171.144,B 90.000,C 0.000} C_DIS
LIN {X 286.543,Y -44.645,Z 74.133,A 171.144,B 90.000,C 0.000} C_DIS
WAIT SEC 1.75
RET=EKI_SetBool("oxy","torchState",TRUE)
RET = EKI_Send("oxy","torchState")
LIN {X 286.175,Y -46.930,Z 73.187,A 170.687,B 90.000,C 0.000} C_DIS
LIN {X 285.791,Y -49.215,Z 72.251,A 170.229,B 90.000,C 0.000} C_DIS
LIN {X 285.388,Y -51.504,Z 71.329,A 169.770,B 90.000,C 0.000} C_DIS
LIN {X 284.965,Y -53.795,Z 70.423,A 169.310,B 90.000,C 0.000} C_DIS
LIN {X 284.523,Y -56.088,Z 69.533,A 168.848,B 90.000,C 0.000} C_DIS
LIN {X 284.061,Y -58.385,Z 68.661,A 168.385,B 90.000,C 0.000} C_DIS
LIN {X 283.579,Y -60.685,Z 67.809,A 167.921,B 90.000,C 0.000} C_DIS
LIN {X 283.076,Y -62.989,Z 66.979,A 167.455,B 90.000,C 0.000} C_DIS
LIN {X 282.552,Y -65.296,Z 66.172,A 166.988,B 90.000,C 0.000} C_DIS
LIN {X 282.008,Y -67.607,Z 65.388,A 166.519,B 90.000,C 0.000} C_DIS
LIN {X 281.444,Y -69.921,Z 64.630,A 166.048,B 90.000,C 0.000} C_DIS
LIN {X 280.857,Y -72.239,Z 63.902,A 165.576,B 90.000,C 0.000} C_DIS
LIN {X 280.251,Y -74.560,Z 63.200,A 165.102,B 90.000,C 0.000} C_DIS
LIN {X 279.621,Y -76.885,Z 62.531,A 164.626,B 90.000,C 0.000} C_DIS
LIN {X 278.971,Y -79.213,Z 61.894,A 164.148,B 90.000,C 0.000} C_DIS
LIN {X 278.298,Y -81.544,Z 61.292,A 163.669,B 90.000,C 0.000} C_DIS
LIN {X 277.605,Y -83.877,Z 60.724,A 163.188,B 90.000,C 0.000} C_DIS
LIN {X 276.888,Y -86.213,Z 60.197,A 162.705,B 90.000,C 0.000} C_DIS
LIN {X 276.150,Y -88.551,Z 59.706,A 162.221,B 90.000,C 0.000} C_DIS
LIN {X 275.388,Y -90.889,Z 59.259,A 161.735,B 90.000,C 0.000} C_DIS
LIN {X 274.605,Y -93.228,Z 58.855,A 161.248,B 90.000,C 0.000} C_DIS
LIN {X 273.800,Y -95.567,Z 58.494,A 160.759,B 90.000,C 0.000} C_DIS
LIN {X 272.973,Y -97.905,Z 58.181,A 160.269,B 90.000,C 0.000} C_DIS
LIN {X 272.124,Y -100.241,Z 57.916,A 159.778,B 90.000,C 0.000} C_DIS
LIN {X 271.448,Y -102.060,Z 57.742,A 159.395,B 90.000,C 0.000} C_DIS
LIN {X 269.576,Y -101.356,Z 57.742,A 159.395,B 90.000,C 0.000} C_DIS
WAIT SEC 0.1
RET=EKI_SetBool("oxy","torchState",FALSE)
RET = EKI_Send("oxy","torchState")
LIN {X 252.727,Y -95.021,Z 57.742,A 159.395,B 90.000,C 0.000} C_DIS
LIN {X 243.072,Y -117.541,Z 81.993,A 154.193,B 90.000,C 0.000} C_DIS
LIN {X 259.277,Y -125.377,Z 81.993,A 154.193,B 90.000,C 0.000} C_DIS
LIN {X 261.077,Y -126.248,Z 81.993,A 154.193,B 90.000,C 0.000} C_DIS
WAIT SEC 1.75
RET=EKI_SetBool("oxy","torchState",TRUE)
RET = EKI_Send("oxy","torchState")
LIN {X 262.145,Y -124.013,Z 82.331,A 154.683,B 90.000,C 0.000} C_DIS
LIN {X 263.193,Y -121.772,Z 82.691,A 155.171,B 90.000,C 0.000} C_DIS
LIN {X 264.220,Y -119.526,Z 83.071,A 155.659,B 90.000,C 0.000} C_DIS
LIN {X 265.228,Y -117.274,Z 83.473,A 156.147,B 90.000,C 0.000} C_DIS
LIN {X 266.215,Y -115.016,Z 83.895,A 156.634,B 90.000,C 0.000} C_DIS
LIN {X 267.182,Y -112.754,Z 84.338,A 157.120,B 90.000,C 0.000} C_DIS
LIN {X 268.127,Y -110.487,Z 84.803,A 157.605,B 90.000,C 0.000} C_DIS
LIN {X 269.051,Y -108.216,Z 85.290,A 158.089,B 90.000,C 0.000} C_DIS
LIN {X 269.954,Y -105.941,Z 85.799,A 158.573,B 90.000,C 0.000} C_DIS
LIN {X 270.837,Y -103.664,Z 86.328,A 159.056,B 90.000,C 0.000} C_DIS
LIN {X 271.700,Y -101.383,Z 86.878,A 159.537,B 90.000,C 0.000} C_DIS
LIN {X 272.542,Y -99.100,Z 87.450,A 160.018,B 90.000,C 0.000} C_DIS
LIN {X 273.361,Y -96.814,Z 88.044,A 160.498,B 90.000,C 0.000} C_DIS
LIN {X 274.160,Y -94.527,Z 88.661,A 160.976,B 90.000,C 0.000} C_DIS
LIN {X 274.938,Y -92.239,Z 89.298,A 161.454,B 90.000,C 0.000} C_DIS
LIN {X 275.696,Y -89.950,Z 89.957,A 161.930,B 90.000,C 0.000} C_DIS
LIN {X 276.433,Y -87.660,Z 90.636,A 162.406,B 90.000,C 0.000} C_DIS
LIN {X 277.149,Y -85.370,Z 91.338,A 162.880,B 90.000,C 0.000} C_DIS
LIN {X 277.843,Y -83.081,Z 92.063,A 163.352,B 90.000,C 0.000} C_DIS
LIN {X 278.517,Y -80.792,Z 92.810,A 163.824,B 90.000,C 0.000} C_DIS
LIN {X 279.170,Y -78.505,Z 93.577,A 164.294,B 90.000,C 0.000} C_DIS
LIN {X 279.804,Y -76.219,Z 94.366,A 164.762,B 90.000,C 0.000} C_DIS
LIN {X 280.417,Y -73.935,Z 95.177,A 165.229,B 90.000,C 0.000} C_DIS
LIN {X 280.779,Y -72.547,Z 95.681,A 165.513,B 90.000,C 0.000} C_DIS
LIN {X 278.843,Y -72.047,Z 95.681,A 165.513,B 90.000,C 0.000} C_DIS
WAIT SEC 0.1
RET=EKI_SetBool("oxy","torchState",FALSE)
RET = EKI_Send("oxy","torchState")
LIN {X 261.415,Y -67.544,Z 95.681,A 165.513,B 90.000,C 0.000} C_DIS
LIN {X 240.991,Y -121.750,Z 108.688,A 153.197,B 90.000,C 0.000} C_DIS
LIN {X 257.057,Y -129.867,Z 108.688,A 153.197,B 90.000,C 0.000} C_DIS
LIN {X 258.843,Y -130.769,Z 108.688,A 153.197,B 90.000,C 0.000} C_DIS
WAIT SEC 1.75
RET=EKI_SetBool("oxy","torchState",TRUE)
RET = EKI_Send("oxy","torchState")
LIN {X 257.724,Y -132.957,Z 108.229,A 152.711,B 90.000,C 0.000} C_DIS
LIN {X 256.588,Y -135.138,Z 107.780,A 152.225,B 90.000,C 0.000} C_DIS
LIN {X 255.431,Y -137.312,Z 107.352,A 151.739,B 90.000,C 0.000} C_DIS
LIN {X 254.254,Y -139.480,Z 106.952,A 151.251,B 90.000,C 0.000} C_DIS
LIN {X 253.054,Y -141.644,Z 106.591,A 150.763,B 90.000,C 0.000} C_DIS
LIN {X 251.834,Y -143.803,Z 106.277,A 150.273,B 90.000,C 0.000} C_DIS
LIN {X 250.592,Y -145.957,Z 106.021,A 149.781,B 90.000,C 0.000} C_DIS
LIN {X 249.328,Y -148.105,Z 105.831,A 149.289,B 90.000,C 0.000} C_DIS
LIN {X 248.044,Y -150.247,Z 105.716,A 148.796,B 90.000,C 0.000} C_DIS
LIN {X 247.381,Y -151.336,Z 105.689,A 148.544,B 90.000,C 0.000} C_DIS
LIN {X 245.675,Y -150.293,Z 105.689,A 148.544,B 90.000,C 0.000} C_DIS
WAIT SEC 0.1
RET=EKI_SetBool("oxy","torchState",FALSE)
RET = EKI_Send("oxy","torchState")
LIN {X 230.320,Y -140.899,Z 105.689,A 148.544,B 90.000,C 0.000} C_DIS
LIN {X 224.145,Y -150.530,Z 105.863,A 146.116,B 90.000,C 0.000} C_DIS
LIN {X 239.088,Y -160.565,Z 105.863,A 146.116,B 90.000,C 0.000} C_DIS
LIN {X 240.748,Y -161.680,Z 105.863,A 146.116,B 90.000,C 0.000} C_DIS
WAIT SEC 1.75
RET=EKI_SetBool("oxy","torchState",TRUE)
RET = EKI_Send("oxy","torchState")
LIN {X 239.346,Y -163.747,Z 105.751,A 145.622,B 90.000,C 0.000} C_DIS
LIN {X 237.931,Y -165.797,Z 105.553,A 145.130,B 90.000,C 0.000} C_DIS
LIN {X 236.501,Y -167.830,Z 105.281,A 144.639,B 90.000,C 0.000} C_DIS
LIN {X 235.059,Y -169.845,Z 104.953,A 144.149,B 90.000,C 0.000} C_DIS
LIN {X 233.602,Y -171.842,Z 104.581,A 143.661,B 90.000,C 0.000} C_DIS
LIN {X 232.131,Y -173.823,Z 104.181,A 143.174,B 90.000,C 0.000} C_DIS
LIN {X 230.643,Y -175.789,Z 103.769,A 142.686,B 90.000,C 0.000} C_DIS
LIN {X 229.141,Y -177.745,Z 103.361,A 142.199,B 90.000,C 0.000} C_DIS
LIN {X 227.621,Y -179.690,Z 102.967,A 141.712,B 90.000,C 0.000} C_DIS
LIN {X 226.080,Y -181.625,Z 102.608,A 141.223,B 90.000,C 0.000} C_DIS
LIN {X 224.518,Y -183.552,Z 102.295,A 140.733,B 90.000,C 0.000} C_DIS
LIN {X 222.936,Y -185.470,Z 102.044,A 140.241,B 90.000,C 0.000} C_DIS
LIN {X 221.405,Y -187.296,Z 101.875,A 139.771,B 90.000,C 0.000} C_DIS
LIN {X 219.878,Y -186.004,Z 101.875,A 139.771,B 90.000,C 0.000} C_DIS
WAIT SEC 0.1
RET=EKI_SetBool("oxy","torchState",FALSE)
RET = EKI_Send("oxy","torchState")
LIN {X 206.136,Y -174.379,Z 101.875,A 139.771,B 90.000,C 0.000} C_DIS
LIN {X 195.155,Y -186.587,Z 101.569,A 136.286,B 90.000,C 0.000} C_DIS
LIN {X 208.165,Y -199.026,Z 101.569,A 136.286,B 90.000,C 0.000} C_DIS
LIN {X 209.611,Y -200.408,Z 101.569,A 136.286,B 90.000,C 0.000} C_DIS
WAIT SEC 1.75
RET=EKI_SetBool("oxy","torchState",TRUE)
RET = EKI_Send("oxy","torchState")
LIN {X 207.883,Y -202.199,Z 101.328,A 135.794,B 90.000,C 0.000} C_DIS
LIN {X 206.148,Y -203.968,Z 101.002,A 135.305,B 90.000,C 0.000} C_DIS
LIN {X 204.403,Y -205.716,Z 100.614,A 134.817,B 90.000,C 0.000} C_DIS
LIN {X 202.649,Y -207.445,Z 100.189,A 134.330,B 90.000,C 0.000} C_DIS
LIN {X 200.882,Y -209.157,Z 99.747,A 133.844,B 90.000,C 0.000} C_DIS
LIN {X 199.098,Y -210.854,Z 99.313,A 133.357,B 90.000,C 0.000} C_DIS
LIN {X 197.298,Y -212.540,Z 98.907,A 132.870,B 90.000,C 0.000} C_DIS
LIN {X 195.477,Y -214.216,Z 98.555,A 132.381,B 90.000,C 0.000} C_DIS
LIN {X 193.635,Y -215.883,Z 98.280,A 131.890,B 90.000,C 0.000} C_DIS
LIN {X 191.772,Y -217.540,Z 98.103,A 131.398,B 90.000,C 0.000} C_DIS
LIN {X 190.651,Y -218.522,Z 98.053,A 131.103,B 90.000,C 0.000} C_DIS
LIN {X 189.337,Y -217.015,Z 98.053,A 131.103,B 90.000,C 0.000} C_DIS
WAIT SEC 0.1
RET=EKI_SetBool("oxy","torchState",FALSE)
RET = EKI_Send("oxy","torchState")
LIN {X 177.503,Y -203.452,Z 98.053,A 131.103,B 90.000,C 0.000} C_DIS
LIN {X 166.771,Y -212.338,Z 97.710,A 128.146,B 90.000,C 0.000} C_DIS
LIN {X 177.889,Y -226.494,Z 97.710,A 128.146,B 90.000,C 0.000} C_DIS
LIN {X 179.124,Y -228.067,Z 97.710,A 128.146,B 90.000,C 0.000} C_DIS
WAIT SEC 1.75
RET=EKI_SetBool("oxy","torchState",TRUE)
RET = EKI_Send("oxy","torchState")
LIN {X 177.214,Y -229.555,Z 97.090,A 127.668,B 90.000,C 0.000} C_DIS
LIN {X 175.324,Y -231.000,Z 96.323,A 127.198,B 90.000,C 0.000} C_DIS
LIN {X 173.428,Y -232.428,Z 95.540,A 126.729,B 90.000,C 0.000} C_DIS
LIN {X 171.493,Y -233.859,Z 94.865,A 126.253,B 90.000,C 0.000} C_DIS
LIN {X 169.500,Y -235.308,Z 94.439,A 125.767,B 90.000,C 0.000} C_DIS
LIN {X 167.469,Y -236.758,Z 94.298,A 125.273,B 90.000,C 0.000} C_DIS
LIN {X 165.422,Y -238.192,Z 94.323,A 124.780,B 90.000,C 0.000} C_DIS
LIN {X 163.363,Y -239.609,Z 94.371,A 124.286,B 90.000,C 0.000} C_DIS
LIN {X 161.292,Y -241.008,Z 94.308,A 123.792,B 90.000,C 0.000} C_DIS
LIN {X 159.225,Y -242.378,Z 93.996,A 123.302,B 90.000,C 0.000} C_DIS
LIN {X 157.191,Y -243.702,Z 93.398,A 122.823,B 90.000,C 0.000} C_DIS
LIN {X 155.194,Y -244.979,Z 92.604,A 122.354,B 90.000,C 0.000} C_DIS
LIN {X 153.219,Y -246.218,Z 91.703,A 121.894,B 90.000,C 0.000} C_DIS
LIN {X 151.240,Y -247.439,Z 90.785,A 121.434,B 90.000,C 0.000} C_DIS
LIN {X 149.229,Y -248.657,Z 89.936,A 120.970,B 90.000,C 0.000} C_DIS
LIN {X 149.129,Y -248.718,Z 89.897,A 120.947,B 90.000,C 0.000} C_DIS
LIN {X 148.101,Y -247.002,Z 89.897,A 120.947,B 90.000,C 0.000} C_DIS
WAIT SEC 0.1
RET=EKI_SetBool("oxy","torchState",FALSE)
RET = EKI_Send("oxy","torchState")
LIN {X 138.845,Y -231.565,Z 89.897,A 120.947,B 90.000,C 0.000} C_DIS
LIN {X 140.790,Y -230.387,Z 113.181,A 121.429,B 90.000,C 0.000} C_DIS
LIN {X 150.176,Y -245.746,Z 113.181,A 121.429,B 90.000,C 0.000} C_DIS
LIN {X 151.219,Y -247.453,Z 113.181,A 121.429,B 90.000,C 0.000} C_DIS
WAIT SEC 1.75
RET=EKI_SetBool("oxy","torchState",TRUE)
RET = EKI_Send("oxy","torchState")
LIN {X 149.096,Y -248.737,Z 112.875,A 120.939,B 90.000,C 0.000} C_DIS
LIN {X 146.967,Y -250.000,Z 112.527,A 120.450,B 90.000,C 0.000} C_DIS
LIN {X 144.830,Y -251.243,Z 112.159,A 119.961,B 90.000,C 0.000} C_DIS
LIN {X 142.683,Y -252.469,Z 111.789,A 119.473,B 90.000,C 0.000} C_DIS
LIN {X 140.525,Y -253.678,Z 111.431,A 118.984,B 90.000,C 0.000} C_DIS
LIN {X 138.351,Y -254.870,Z 111.108,A 118.495,B 90.000,C 0.000} C_DIS
LIN {X 136.162,Y -256.046,Z 110.837,A 118.004,B 90.000,C 0.000} C_DIS
LIN {X 133.957,Y -257.207,Z 110.638,A 117.511,B 90.000,C 0.000} C_DIS
LIN {X 131.737,Y -258.351,Z 110.530,A 117.018,B 90.000,C 0.000} C_DIS
LIN {X 129.930,Y -259.265,Z 110.521,A 116.618,B 90.000,C 0.000} C_DIS
LIN {X 129.034,Y -257.477,Z 110.521,A 116.618,B 90.000,C 0.000} C_DIS
WAIT SEC 0.1
RET=EKI_SetBool("oxy","torchState",FALSE)
RET = EKI_Send("oxy","torchState")
LIN {X 120.970,Y -241.384,Z 110.521,A 116.618,B 90.000,C 0.000} C_DIS
LIN {X 110.855,Y -246.193,Z 112.573,A 114.241,B 90.000,C 0.000} C_DIS
LIN {X 118.246,Y -262.606,Z 112.573,A 114.241,B 90.000,C 0.000} C_DIS
LIN {X 119.067,Y -264.430,Z 112.573,A 114.241,B 90.000,C 0.000} C_DIS
WAIT SEC 1.75
RET=EKI_SetBool("oxy","torchState",TRUE)
RET = EKI_Send("oxy","torchState")
LIN {X 116.963,Y -265.367,Z 113.544,A 113.786,B 90.000,C 0.000} C_DIS
LIN {X 114.945,Y -266.247,Z 114.728,A 113.351,B 90.000,C 0.000} C_DIS
LIN {X 113.041,Y -267.061,Z 116.128,A 112.942,B 90.000,C 0.000} C_DIS
LIN {X 111.283,Y -267.799,Z 117.746,A 112.565,B 90.000,C 0.000} C_DIS
LIN {X 109.854,Y -268.388,Z 119.389,A 112.260,B 90.000,C 0.000} C_DIS
LIN {X 109.097,Y -266.537,Z 119.389,A 112.260,B 90.000,C 0.000} C_DIS
WAIT SEC 0.1
RET=EKI_SetBool("oxy","torchState",FALSE)
RET = EKI_Send("oxy","torchState")
LIN {X 102.278,Y -249.878,Z 119.389,A 112.260,B 90.000,C 0.000} C_DIS
LIN {X 97.299,Y -251.859,Z 134.611,A 111.123,B 90.000,C 0.000} C_DIS
LIN {X 103.786,Y -268.649,Z 134.611,A 111.123,B 90.000,C 0.000} C_DIS
LIN {X 104.507,Y -270.515,Z 134.611,A 111.123,B 90.000,C 0.000} C_DIS
WAIT SEC 1.75
RET=EKI_SetBool("oxy","torchState",TRUE)
RET = EKI_Send("oxy","torchState")
LIN {X 104.341,Y -270.579,Z 137.104,A 111.088,B 90.000,C 0.000} C_DIS
LIN {X 104.287,Y -270.600,Z 139.603,A 111.076,B 90.000,C 0.000} C_DIS
LIN {X 104.318,Y -270.588,Z 142.103,A 111.083,B 90.000,C 0.000} C_DIS
LIN {X 104.410,Y -270.552,Z 144.601,A 111.102,B 90.000,C 0.000} C_DIS
LIN {X 104.543,Y -270.501,Z 147.096,A 111.131,B 90.000,C 0.000} C_DIS
LIN {X 104.690,Y -270.444,Z 149.591,A 111.162,B 90.000,C 0.000} C_DIS
LIN {X 104.779,Y -270.410,Z 151.113,A 111.181,B 90.000,C 0.000} C_DIS
LIN {X 104.057,Y -268.545,Z 151.113,A 111.181,B 90.000,C 0.000} C_DIS
WAIT SEC 0.1
RET=EKI_SetBool("oxy","torchState",FALSE)
RET = EKI_Send("oxy","torchState")
LIN {X 97.553,Y -251.761,Z 151.113,A 111.181,B 90.000,C 0.000} C_DIS
LIN {X 120.985,Y -241.377,Z 159.512,A 116.621,B 90.000,C 0.000} C_DIS
LIN {X 129.051,Y -257.468,Z 159.512,A 116.621,B 90.000,C 0.000} C_DIS
LIN {X 129.947,Y -259.256,Z 159.512,A 116.621,B 90.000,C 0.000} C_DIS
WAIT SEC 1.75
RET=EKI_SetBool("oxy","torchState",TRUE)
RET = EKI_Send("oxy","torchState")
LIN {X 130.115,Y -259.172,Z 157.020,A 116.658,B 90.000,C 0.000} C_DIS
LIN {X 130.402,Y -259.028,Z 154.541,A 116.722,B 90.000,C 0.000} C_DIS
LIN {X 130.830,Y -258.812,Z 152.087,A 116.817,B 90.000,C 0.000} C_DIS
LIN {X 131.422,Y -258.511,Z 149.678,A 116.948,B 90.000,C 0.000} C_DIS
LIN {X 132.193,Y -258.118,Z 147.332,A 117.119,B 90.000,C 0.000} C_DIS
LIN {X 132.622,Y -257.898,Z 146.260,A 117.214,B 90.000,C 0.000} C_DIS
LIN {X 131.707,Y -256.120,Z 146.260,A 117.214,B 90.000,C 0.000} C_DIS
WAIT SEC 0.1
RET=EKI_SetBool("oxy","torchState",FALSE)
RET = EKI_Send("oxy","torchState")
LIN {X 123.475,Y -240.112,Z 146.260,A 117.214,B 90.000,C 0.000} C_DIS
LIN {X 131.153,Y -236.006,Z 136.669,A 119.062,B 90.000,C 0.000} C_DIS
LIN {X 139.896,Y -251.740,Z 136.669,A 119.062,B 90.000,C 0.000} C_DIS
LIN {X 140.868,Y -253.488,Z 136.669,A 119.062,B 90.000,C 0.000} C_DIS
WAIT SEC 1.75
RET=EKI_SetBool("oxy","torchState",TRUE)
RET = EKI_Send("oxy","torchState")
LIN {X 142.918,Y -252.338,Z 135.821,A 119.526,B 90.000,C 0.000} C_DIS
LIN {X 145.037,Y -251.126,Z 135.280,A 120.008,B 90.000,C 0.000} C_DIS
LIN {X 147.181,Y -249.875,Z 134.983,A 120.499,B 90.000,C 0.000} C_DIS
LIN {X 149.326,Y -248.599,Z 134.850,A 120.992,B 90.000,C 0.000} C_DIS
LIN {X 151.463,Y -247.303,Z 134.809,A 121.486,B 90.000,C 0.000} C_DIS
LIN {X 153.589,Y -245.988,Z 134.793,A 121.980,B 90.000,C 0.000} C_DIS
LIN {X 153.732,Y -245.899,Z 134.792,A 122.013,B 90.000,C 0.000} C_DIS
LIN {X 152.672,Y -244.203,Z 134.792,A 122.013,B 90.000,C 0.000} C_DIS
WAIT SEC 0.1
RET=EKI_SetBool("oxy","torchState",FALSE)
RET = EKI_Send("oxy","torchState")
LIN {X 143.130,Y -228.941,Z 134.792,A 122.013,B 90.000,C 0.000} C_DIS
LIN {X 155.965,Y -220.397,Z 134.558,A 125.285,B 90.000,C 0.000} C_DIS
LIN {X 166.363,Y -235.090,Z 134.558,A 125.285,B 90.000,C 0.000} C_DIS
LIN {X 167.518,Y -236.723,Z 134.558,A 125.285,B 90.000,C 0.000} C_DIS
WAIT SEC 1.75
RET=EKI_SetBool("oxy","torchState",TRUE)
RET = EKI_Send("oxy","torchState")
LIN {X 169.546,Y -235.274,Z 134.749,A 125.778,B 90.000,C 0.000} C_DIS
LIN {X 171.554,Y -233.814,Z 135.044,A 126.268,B 90.000,C 0.000} C_DIS
LIN {X 173.537,Y -232.346,Z 135.445,A 126.756,B 90.000,C 0.000} C_DIS
LIN {X 175.492,Y -230.873,Z 135.952,A 127.239,B 90.000,C 0.000} C_DIS
LIN {X 177.416,Y -229.398,Z 136.561,A 127.718,B 90.000,C 0.000} C_DIS
LIN {X 179.305,Y -227.925,Z 137.276,A 128.192,B 90.000,C 0.000} C_DIS
LIN {X 181.156,Y -226.456,Z 138.090,A 128.658,B 90.000,C 0.000} C_DIS
LIN {X 182.966,Y -224.996,Z 139.009,A 129.118,B 90.000,C 0.000} C_DIS
LIN {X 184.731,Y -223.549,Z 140.027,A 129.569,B 90.000,C 0.000} C_DIS
LIN {X 186.450,Y -222.118,Z 141.144,A 130.011,B 90.000,C 0.000} C_DIS
LIN {X 188.116,Y -220.709,Z 142.363,A 130.442,B 90.000,C 0.000} C_DIS
LIN {X 189.729,Y -219.323,Z 143.677,A 130.862,B 90.000,C 0.000} C_DIS
LIN {X 189.952,Y -219.130,Z 143.869,A 130.920,B 90.000,C 0.000} C_DIS
LIN {X 188.642,Y -217.619,Z 143.869,A 130.920,B 90.000,C 0.000} C_DIS
WAIT SEC 0.1
RET=EKI_SetBool("oxy","torchState",FALSE)
RET = EKI_Send("oxy","torchState")
LIN {X 176.852,Y -204.018,Z 143.869,A 130.920,B 90.000,C 0.000} C_DIS
LIN {X 184.010,Y -197.586,Z 122.905,A 132.962,B 90.000,C 0.000} C_DIS
LIN {X 196.277,Y -210.759,Z 122.905,A 132.962,B 90.000,C 0.000} C_DIS
LIN {X 197.640,Y -212.222,Z 122.905,A 132.962,B 90.000,C 0.000} C_DIS
WAIT SEC 1.75
RET=EKI_SetBool("oxy","torchState",TRUE)
RET = EKI_Send("oxy","torchState")
LIN {X 196.058,Y -213.685,Z 121.638,A 132.537,B 90.000,C 0.000} C_DIS
LIN {X 194.413,Y -215.183,Z 120.498,A 132.097,B 90.000,C 0.000} C_DIS
LIN {X 192.712,Y -216.707,Z 119.482,A 131.646,B 90.000,C 0.000} C_DIS
LIN {X 190.962,Y -218.250,Z 118.584,A 131.185,B 90.000,C 0.000} C_DIS
LIN {X 189.170,Y -219.805,Z 117.798,A 130.716,B 90.000,C 0.000} C_DIS
LIN {X 187.341,Y -221.367,Z 117.117,A 130.241,B 90.000,C 0.000} C_DIS
LIN {X 185.480,Y -222.929,Z 116.530,A 129.761,B 90.000,C 0.000} C_DIS
LIN {X 183.590,Y -224.487,Z 116.032,A 129.277,B 90.000,C 0.000} C_DIS
LIN {X 181.675,Y -226.039,Z 115.615,A 128.790,B 90.000,C 0.000} C_DIS
LIN {X 179.739,Y -227.582,Z 115.268,A 128.301,B 90.000,C 0.000} C_DIS
LIN {X 177.783,Y -229.113,Z 114.987,A 127.810,B 90.000,C 0.000} C_DIS
LIN {X 175.868,Y -230.587,Z 114.766,A 127.333,B 90.000,C 0.000} C_DIS
LIN {X 174.655,Y -228.997,Z 114.766,A 127.333,B 90.000,C 0.000} C_DIS
WAIT SEC 0.1
RET=EKI_SetBool("oxy","torchState",FALSE)
RET = EKI_Send("oxy","torchState")
LIN {X 163.739,Y -214.685,Z 114.766,A 127.333,B 90.000,C 0.000} C_DIS
LIN {X 171.905,Y -208.203,Z 76.278,A 129.545,B 90.000,C 0.000} C_DIS
LIN {X 183.365,Y -222.084,Z 76.278,A 129.545,B 90.000,C 0.000} C_DIS
LIN {X 184.639,Y -223.626,Z 76.278,A 129.545,B 90.000,C 0.000} C_DIS
WAIT SEC 1.75
RET=EKI_SetBool("oxy","torchState",TRUE)
RET = EKI_Send("oxy","torchState")
LIN {X 186.509,Y -222.069,Z 76.848,A 130.026,B 90.000,C 0.000} C_DIS
LIN {X 188.356,Y -220.503,Z 77.469,A 130.504,B 90.000,C 0.000} C_DIS
LIN {X 190.184,Y -218.928,Z 78.121,A 130.981,B 90.000,C 0.000} C_DIS
LIN {X 191.994,Y -217.340,Z 78.792,A 131.457,B 90.000,C 0.000} C_DIS
LIN {X 193.791,Y -215.739,Z 79.468,A 131.932,B 90.000,C 0.000} C_DIS
LIN {X 195.578,Y -214.123,Z 80.134,A 132.408,B 90.000,C 0.000} C_DIS
LIN {X 197.356,Y -212.487,Z 80.775,A 132.886,B 90.000,C 0.000} C_DIS
LIN {X 199.127,Y -210.828,Z 81.375,A 133.365,B 90.000,C 0.000} C_DIS
LIN {X 200.894,Y -209.145,Z 81.919,A 133.847,B 90.000,C 0.000} C_DIS
LIN {X 202.657,Y -207.437,Z 82.393,A 134.332,B 90.000,C 0.000} C_DIS
LIN {X 204.416,Y -205.704,Z 82.778,A 134.820,B 90.000,C 0.000} C_DIS
LIN {X 206.170,Y -203.946,Z 83.064,A 135.311,B 90.000,C 0.000} C_DIS
LIN {X 207.915,Y -202.166,Z 83.251,A 135.803,B 90.000,C 0.000} C_DIS
LIN {X 209.649,Y -200.368,Z 83.350,A 136.297,B 90.000,C 0.000} C_DIS
LIN {X 211.368,Y -198.553,Z 83.366,A 136.791,B 90.000,C 0.000} C_DIS
LIN {X 213.071,Y -196.725,Z 83.311,A 137.284,B 90.000,C 0.000} C_DIS
LIN {X 214.757,Y -194.883,Z 83.195,A 137.778,B 90.000,C 0.000} C_DIS
LIN {X 216.425,Y -193.029,Z 83.026,A 138.270,B 90.000,C 0.000} C_DIS
LIN {X 218.074,Y -191.162,Z 82.811,A 138.762,B 90.000,C 0.000} C_DIS
LIN {X 219.707,Y -189.285,Z 82.565,A 139.254,B 90.000,C 0.000} C_DIS
LIN {X 221.319,Y -187.395,Z 82.290,A 139.745,B 90.000,C 0.000} C_DIS
LIN {X 222.915,Y -185.493,Z 82.001,A 140.235,B 90.000,C 0.000} C_DIS
LIN {X 224.495,Y -183.579,Z 81.704,A 140.726,B 90.000,C 0.000} C_DIS
LIN {X 226.059,Y -181.651,Z 81.406,A 141.216,B 90.000,C 0.000} C_DIS
LIN {X 227.606,Y -179.709,Z 81.119,A 141.707,B 90.000,C 0.000} C_DIS
LIN {X 228.946,Y -178.000,Z 80.882,A 142.136,B 90.000,C 0.000} C_DIS
LIN {X 227.367,Y -176.772,Z 80.882,A 142.136,B 90.000,C 0.000} C_DIS
WAIT SEC 0.1
RET=EKI_SetBool("oxy","torchState",FALSE)
RET = EKI_Send("oxy","torchState")
LIN {X 213.156,Y -165.724,Z 80.882,A 142.136,B 90.000,C 0.000} C_DIS
LIN {X 229.941,Y -141.518,Z 60.139,A 148.390,B 90.000,C 0.000} C_DIS
LIN {X 245.270,Y -150.952,Z 60.139,A 148.390,B 90.000,C 0.000} C_DIS
LIN {X 246.973,Y -152.000,Z 60.139,A 148.390,B 90.000,C 0.000} C_DIS
WAIT SEC 1.75
RET=EKI_SetBool("oxy","torchState",TRUE)
RET = EKI_Send("oxy","torchState")
LIN {X 245.654,Y -154.119,Z 60.281,A 147.897,B 90.000,C 0.000} C_DIS
LIN {X 244.318,Y -156.228,Z 60.406,A 147.403,B 90.000,C 0.000} C_DIS
LIN {X 242.964,Y -158.326,Z 60.513,A 146.910,B 90.000,C 0.000} C_DIS
LIN {X 241.591,Y -160.413,Z 60.601,A 146.416,B 90.000,C 0.000} C_DIS
LIN {X 240.200,Y -162.489,Z 60.671,A 145.923,B 90.000,C 0.000} C_DIS
LIN {X 238.791,Y -164.553,Z 60.724,A 145.429,B 90.000,C 0.000} C_DIS
LIN {X 237.364,Y -166.605,Z 60.759,A 144.935,B 90.000,C 0.000} C_DIS
LIN {X 235.919,Y -168.645,Z 60.777,A 144.441,B 90.000,C 0.000} C_DIS
LIN {X 234.457,Y -170.672,Z 60.778,A 143.947,B 90.000,C 0.000} C_DIS
LIN {X 232.977,Y -172.687,Z 60.762,A 143.453,B 90.000,C 0.000} C_DIS
LIN {X 231.480,Y -174.688,Z 60.730,A 142.960,B 90.000,C 0.000} C_DIS
LIN {X 229.965,Y -176.677,Z 60.683,A 142.466,B 90.000,C 0.000} C_DIS
LIN {X 228.434,Y -178.652,Z 60.619,A 141.972,B 90.000,C 0.000} C_DIS
LIN {X 226.887,Y -180.613,Z 60.541,A 141.478,B 90.000,C 0.000} C_DIS
LIN {X 225.322,Y -182.561,Z 60.447,A 140.985,B 90.000,C 0.000} C_DIS
LIN {X 223.742,Y -184.494,Z 60.339,A 140.492,B 90.000,C 0.000} C_DIS
LIN {X 222.145,Y -186.413,Z 60.217,A 139.998,B 90.000,C 0.000} C_DIS
LIN {X 220.532,Y -188.318,Z 60.080,A 139.505,B 90.000,C 0.000} C_DIS
LIN {X 218.904,Y -190.209,Z 59.931,A 139.012,B 90.000,C 0.000} C_DIS
LIN {X 217.260,Y -192.085,Z 59.768,A 138.519,B 90.000,C 0.000} C_DIS
LIN {X 215.601,Y -193.947,Z 59.593,A 138.027,B 90.000,C 0.000} C_DIS
LIN {X 213.927,Y -195.794,Z 59.406,A 137.534,B 90.000,C 0.000} C_DIS
LIN {X 212.236,Y -197.623,Z 59.204,A 137.042,B 90.000,C 0.000} C_DIS
LIN {X 210.530,Y -199.438,Z 58.991,A 136.550,B 90.000,C 0.000} C_DIS
LIN {X 208.809,Y -201.237,Z 58.767,A 136.058,B 90.000,C 0.000} C_DIS
LIN {X 207.075,Y -203.022,Z 58.532,A 135.566,B 90.000,C 0.000} C_DIS
LIN {X 205.326,Y -204.792,Z 58.286,A 135.075,B 90.000,C 0.000} C_DIS
LIN {X 203.565,Y -206.547,Z 58.031,A 134.583,B 90.000,C 0.000} C_DIS
LIN {X 202.161,Y -205.122,Z 58.031,A 134.583,B 90.000,C 0.000} C_DIS
WAIT SEC 0.1
RET=EKI_SetBool("oxy","torchState",FALSE)
RET = EKI_Send("oxy","torchState")
LIN {X 189.526,Y -192.302,Z 58.031,A 134.583,B 90.000,C 0.000} C_DIS
LIN {X 141.617,Y -229.880,Z 48.543,A 121.635,B 90.000,C 0.000} C_DIS
LIN {X 151.058,Y -245.205,Z 48.543,A 121.635,B 90.000,C 0.000} C_DIS
LIN {X 152.107,Y -246.908,Z 48.543,A 121.635,B 90.000,C 0.000} C_DIS
WAIT SEC 1.75
RET=EKI_SetBool("oxy","torchState",TRUE)
RET = EKI_Send("oxy","torchState")
LIN {X 150.001,Y -248.188,Z 48.125,A 121.148,B 90.000,C 0.000} C_DIS
LIN {X 147.886,Y -249.453,Z 47.706,A 120.661,B 90.000,C 0.000} C_DIS
LIN {X 145.762,Y -250.703,Z 47.287,A 120.174,B 90.000,C 0.000} C_DIS
LIN {X 143.626,Y -251.932,Z 46.867,A 119.687,B 90.000,C 0.000} C_DIS
LIN {X 141.480,Y -253.141,Z 46.446,A 119.201,B 90.000,C 0.000} C_DIS
LIN {X 139.324,Y -254.336,Z 46.026,A 118.714,B 90.000,C 0.000} C_DIS
LIN {X 137.159,Y -255.512,Z 45.606,A 118.227,B 90.000,C 0.000} C_DIS
LIN {X 134.983,Y -256.670,Z 45.186,A 117.740,B 90.000,C 0.000} C_DIS
LIN {X 132.797,Y -257.806,Z 44.766,A 117.253,B 90.000,C 0.000} C_DIS
LIN {X 130.600,Y -258.923,Z 44.349,A 116.766,B 90.000,C 0.000} C_DIS
LIN {X 128.395,Y -260.024,Z 43.933,A 116.279,B 90.000,C 0.000} C_DIS
LIN {X 126.181,Y -261.109,Z 43.517,A 115.792,B 90.000,C 0.000} C_DIS
LIN {X 123.957,Y -262.172,Z 43.106,A 115.305,B 90.000,C 0.000} C_DIS
LIN {X 121.723,Y -263.215,Z 42.695,A 114.818,B 90.000,C 0.000} C_DIS
LIN {X 119.479,Y -264.241,Z 42.289,A 114.331,B 90.000,C 0.000} C_DIS
LIN {X 117.227,Y -265.247,Z 41.884,A 113.843,B 90.000,C 0.000} C_DIS
LIN {X 114.964,Y -266.230,Z 41.484,A 113.356,B 90.000,C 0.000} C_DIS
LIN {X 112.695,Y -267.201,Z 41.086,A 112.868,B 90.000,C 0.000} C_DIS
LIN {X 110.416,Y -268.149,Z 40.694,A 112.380,B 90.000,C 0.000} C_DIS
LIN {X 108.131,Y -269.084,Z 40.304,A 111.893,B 90.000,C 0.000} C_DIS
LIN {X 105.833,Y -269.991,Z 39.922,A 111.405,B 90.000,C 0.000} C_DIS
LIN {X 103.819,Y -270.779,Z 39.588,A 110.977,B 90.000,C 0.000} C_DIS
LIN {X 103.103,Y -268.912,Z 39.588,A 110.977,B 90.000,C 0.000} C_DIS
WAIT SEC 0.1
RET=EKI_SetBool("oxy","torchState",FALSE)
RET = EKI_Send("oxy","torchState")
LIN {X 96.659,Y -252.105,Z 39.588,A 110.977,B 90.000,C 0.000} C_DIS
LIN {X 94.744,Y -252.831,Z 59.460,A 110.543,B 90.000,C 0.000} C_DIS
LIN {X 101.060,Y -269.686,Z 59.460,A 110.543,B 90.000,C 0.000} C_DIS
LIN {X 101.762,Y -271.559,Z 59.460,A 110.543,B 90.000,C 0.000} C_DIS
WAIT SEC 1.75
RET=EKI_SetBool("oxy","torchState",TRUE)
RET = EKI_Send("oxy","torchState")
LIN {X 103.998,Y -270.711,Z 60.188,A 111.015,B 90.000,C 0.000} C_DIS
LIN {X 106.210,Y -269.851,Z 60.973,A 111.484,B 90.000,C 0.000} C_DIS
LIN {X 108.400,Y -268.977,Z 61.803,A 111.950,B 90.000,C 0.000} C_DIS
LIN {X 110.575,Y -268.092,Z 62.661,A 112.414,B 90.000,C 0.000} C_DIS
LIN {X 112.735,Y -267.189,Z 63.538,A 112.876,B 90.000,C 0.000} C_DIS
LIN {X 114.885,Y -266.267,Z 64.417,A 113.339,B 90.000,C 0.000} C_DIS
LIN {X 117.034,Y -265.336,Z 65.292,A 113.801,B 90.000,C 0.000} C_DIS
LIN {X 119.180,Y -264.378,Z 66.143,A 114.266,B 90.000,C 0.000} C_DIS
LIN {X 121.330,Y -263.399,Z 66.960,A 114.732,B 90.000,C 0.000} C_DIS
LIN {X 123.486,Y -262.394,Z 67.728,A 115.202,B 90.000,C 0.000} C_DIS
LIN {X 125.350,Y -261.510,Z 68.343,A 115.610,B 90.000,C 0.000} C_DIS
LIN {X 124.486,Y -259.706,Z 68.343,A 115.610,B 90.000,C 0.000} C_DIS
WAIT SEC 0.1
RET=EKI_SetBool("oxy","torchState",FALSE)
RET = EKI_Send("oxy","torchState")
LIN {X 116.705,Y -243.475,Z 68.343,A 115.610,B 90.000,C 0.000} C_DIS
LIN {X 111.528,Y -245.889,Z 88.699,A 114.398,B 90.000,C 0.000} C_DIS
LIN {X 118.963,Y -262.282,Z 88.699,A 114.398,B 90.000,C 0.000} C_DIS
LIN {X 119.789,Y -264.103,Z 88.699,A 114.398,B 90.000,C 0.000} C_DIS
WAIT SEC 1.75
RET=EKI_SetBool("oxy","torchState",TRUE)
RET = EKI_Send("oxy","torchState")
LIN {X 117.512,Y -265.123,Z 88.840,A 113.905,B 90.000,C 0.000} C_DIS
LIN {X 115.224,Y -266.126,Z 88.951,A 113.411,B 90.000,C 0.000} C_DIS
LIN {X 112.927,Y -267.108,Z 89.030,A 112.918,B 90.000,C 0.000} C_DIS
LIN {X 110.621,Y -268.072,Z 88.977,A 112.424,B 90.000,C 0.000} C_DIS
LIN {X 108.310,Y -269.014,Z 88.843,A 111.931,B 90.000,C 0.000} C_DIS
LIN {X 105.993,Y -269.935,Z 88.672,A 111.438,B 90.000,C 0.000} C_DIS
LIN {X 103.670,Y -270.836,Z 88.464,A 110.946,B 90.000,C 0.000} C_DIS
LIN {X 101.343,Y -271.715,Z 88.219,A 110.454,B 90.000,C 0.000} C_DIS
LIN {X 99.012,Y -272.573,Z 87.937,A 109.964,B 90.000,C 0.000} C_DIS
LIN {X 96.678,Y -273.410,Z 87.618,A 109.474,B 90.000,C 0.000} C_DIS
LIN {X 94.342,Y -274.225,Z 87.264,A 108.985,B 90.000,C 0.000} C_DIS
LIN {X 92.004,Y -275.018,Z 86.871,A 108.497,B 90.000,C 0.000} C_DIS
LIN {X 91.009,Y -275.349,Z 86.695,A 108.290,B 90.000,C 0.000} C_DIS
LIN {X 90.382,Y -273.450,Z 86.695,A 108.290,B 90.000,C 0.000} C_DIS
WAIT SEC 0.1
RET=EKI_SetBool("oxy","torchState",FALSE)
RET = EKI_Send("oxy","torchState")
LIN {X 84.733,Y -256.360,Z 86.695,A 108.290,B 90.000,C 0.000} C_DIS
LIN {X 6.140,Y -269.930,Z 102.178,A 91.303,B 90.000,C 0.000} C_DIS
LIN {X 6.549,Y -287.926,Z 102.178,A 91.303,B 90.000,C 0.000} C_DIS
LIN {X 6.595,Y -289.925,Z 102.178,A 91.303,B 90.000,C 0.000} C_DIS
WAIT SEC 1.75
RET=EKI_SetBool("oxy","torchState",TRUE)
RET = EKI_Send("oxy","torchState")
LIN {X 4.125,Y -289.970,Z 101.795,A 90.815,B 90.000,C 0.000} C_DIS
LIN {X 1.698,Y -289.995,Z 101.198,A 90.336,B 90.000,C 0.000} C_DIS
LIN {X -0.656,Y -289.999,Z 100.358,A 89.870,B 90.000,C 0.000} C_DIS
LIN {X -2.896,Y -289.985,Z 99.248,A 89.428,B 90.000,C 0.000} C_DIS
LIN {X -4.965,Y -289.957,Z 97.845,A 89.019,B 90.000,C 0.000} C_DIS
LIN {X -6.800,Y -289.920,Z 96.149,A 88.656,B 90.000,C 0.000} C_DIS
LIN {X -8.342,Y -289.880,Z 94.182,A 88.352,B 90.000,C 0.000} C_DIS
LIN {X -9.519,Y -289.844,Z 91.977,A 88.119,B 90.000,C 0.000} C_DIS
LIN {X -10.194,Y -289.821,Z 89.835,A 87.985,B 90.000,C 0.000} C_DIS
LIN {X -10.124,Y -287.822,Z 89.835,A 87.985,B 90.000,C 0.000} C_DIS
WAIT SEC 0.1
RET=EKI_SetBool("oxy","torchState",FALSE)
RET = EKI_Send("oxy","torchState")
LIN {X -9.491,Y -269.833,Z 89.835,A 87.985,B 90.000,C 0.000} C_DIS
LIN {X 120.692,Y -241.523,Z 186.817,A 116.552,B 90.000,C 0.000} C_DIS
LIN {X 128.738,Y -257.625,Z 186.817,A 116.552,B 90.000,C 0.000} C_DIS
LIN {X 129.632,Y -259.414,Z 186.817,A 116.552,B 90.000,C 0.000} C_DIS
WAIT SEC 1.75
RET=EKI_SetBool("oxy","torchState",TRUE)
RET = EKI_Send("oxy","torchState")
LIN {X 129.155,Y -259.651,Z 189.259,A 116.447,B 90.000,C 0.000} C_DIS
LIN {X 128.542,Y -259.956,Z 191.663,A 116.311,B 90.000,C 0.000} C_DIS
LIN {X 127.801,Y -260.321,Z 194.023,A 116.148,B 90.000,C 0.000} C_DIS
LIN {X 126.947,Y -260.738,Z 196.334,A 115.960,B 90.000,C 0.000} C_DIS
LIN {X 125.990,Y -261.202,Z 198.597,A 115.750,B 90.000,C 0.000} C_DIS
LIN {X 124.944,Y -261.704,Z 200.811,A 115.521,B 90.000,C 0.000} C_DIS
LIN {X 123.822,Y -262.237,Z 202.980,A 115.276,B 90.000,C 0.000} C_DIS
LIN {X 122.635,Y -262.794,Z 205.108,A 115.016,B 90.000,C 0.000} C_DIS
LIN {X 121.392,Y -263.370,Z 207.199,A 114.746,B 90.000,C 0.000} C_DIS
LIN {X 120.105,Y -263.959,Z 209.259,A 114.466,B 90.000,C 0.000} C_DIS
LIN {X 118.783,Y -264.557,Z 211.295,A 114.179,B 90.000,C 0.000} C_DIS
LIN {X 117.433,Y -265.159,Z 213.311,A 113.887,B 90.000,C 0.000} C_DIS
LIN {X 116.063,Y -265.762,Z 215.313,A 113.592,B 90.000,C 0.000} C_DIS
LIN {X 114.683,Y -266.360,Z 217.309,A 113.295,B 90.000,C 0.000} C_DIS
LIN {X 114.489,Y -266.444,Z 217.589,A 113.253,B 90.000,C 0.000} C_DIS
LIN {X 113.699,Y -264.606,Z 217.589,A 113.253,B 90.000,C 0.000} C_DIS
WAIT SEC 0.1
RET=EKI_SetBool("oxy","torchState",FALSE)
RET = EKI_Send("oxy","torchState")
LIN {X 106.593,Y -248.068,Z 217.589,A 113.253,B 90.000,C 0.000} C_DIS
LIN {X 128.856,Y -237.268,Z 223.745,A 118.505,B 90.000,C 0.000} C_DIS
LIN {X 137.446,Y -253.086,Z 223.745,A 118.505,B 90.000,C 0.000} C_DIS
LIN {X 138.400,Y -254.844,Z 223.745,A 118.505,B 90.000,C 0.000} C_DIS
WAIT SEC 1.75
RET=EKI_SetBool("oxy","torchState",TRUE)
RET = EKI_Send("oxy","torchState")
LIN {X 139.457,Y -254.267,Z 221.554,A 118.743,B 90.000,C 0.000} C_DIS
LIN {X 140.501,Y -253.691,Z 219.356,A 118.979,B 90.000,C 0.000} C_DIS
LIN {X 141.531,Y -253.118,Z 217.152,A 119.212,B 90.000,C 0.000} C_DIS
LIN {X 142.548,Y -252.547,Z 214.942,A 119.442,B 90.000,C 0.000} C_DIS
LIN {X 143.551,Y -251.978,Z 212.724,A 119.670,B 90.000,C 0.000} C_DIS
LIN {X 144.541,Y -251.411,Z 210.500,A 119.895,B 90.000,C 0.000} C_DIS
LIN {X 145.518,Y -250.847,Z 208.269,A 120.118,B 90.000,C 0.000} C_DIS
LIN {X 146.481,Y -250.286,Z 206.032,A 120.339,B 90.000,C 0.000} C_DIS
LIN {X 147.431,Y -249.727,Z 203.788,A 120.556,B 90.000,C 0.000} C_DIS
LIN {X 148.368,Y -249.172,Z 201.538,A 120.771,B 90.000,C 0.000} C_DIS
LIN {X 149.292,Y -248.620,Z 199.282,A 120.984,B 90.000,C 0.000} C_DIS
LIN {X 150.202,Y -248.071,Z 197.019,A 121.194,B 90.000,C 0.000} C_DIS
LIN {X 150.898,Y -247.649,Z 195.267,A 121.355,B 90.000,C 0.000} C_DIS
LIN {X 149.857,Y -245.941,Z 195.267,A 121.355,B 90.000,C 0.000} C_DIS
WAIT SEC 0.1
RET=EKI_SetBool("oxy","torchState",FALSE)
RET = EKI_Send("oxy","torchState")
LIN {X 140.491,Y -230.569,Z 195.267,A 121.355,B 90.000,C 0.000} C_DIS
LIN {X 142.554,Y -229.300,Z 172.563,A 121.869,B 90.000,C 0.000} C_DIS
LIN {X 152.058,Y -244.586,Z 172.563,A 121.869,B 90.000,C 0.000} C_DIS
LIN {X 153.113,Y -246.285,Z 172.563,A 121.869,B 90.000,C 0.000} C_DIS
WAIT SEC 1.75
RET=EKI_SetBool("oxy","torchState",TRUE)
RET = EKI_Send("oxy","torchState")
LIN {X 155.087,Y -245.045,Z 171.660,A 122.329,B 90.000,C 0.000} C_DIS
LIN {X 157.050,Y -243.789,Z 170.756,A 122.790,B 90.000,C 0.000} C_DIS
LIN {X 159.005,Y -242.519,Z 169.852,A 123.250,B 90.000,C 0.000} C_DIS
LIN {X 160.949,Y -241.234,Z 168.948,A 123.711,B 90.000,C 0.000} C_DIS
LIN {X 162.883,Y -239.934,Z 168.045,A 124.171,B 90.000,C 0.000} C_DIS
LIN {X 164.806,Y -238.617,Z 167.141,A 124.632,B 90.000,C 0.000} C_DIS
LIN {X 166.718,Y -237.284,Z 166.237,A 125.092,B 90.000,C 0.000} C_DIS
LIN {X 167.442,Y -236.777,Z 165.894,A 125.267,B 90.000,C 0.000} C_DIS
LIN {X 166.287,Y -235.144,Z 165.894,A 125.267,B 90.000,C 0.000} C_DIS
WAIT SEC 0.1
RET=EKI_SetBool("oxy","torchState",FALSE)
RET = EKI_Send("oxy","torchState")
LIN {X 155.894,Y -220.447,Z 165.894,A 125.267,B 90.000,C 0.000} C_DIS
LIN {X 167.461,Y -211.794,Z 174.604,A 128.333,B 90.000,C 0.000} C_DIS
LIN {X 178.625,Y -225.914,Z 174.604,A 128.333,B 90.000,C 0.000} C_DIS
LIN {X 179.866,Y -227.483,Z 174.604,A 128.333,B 90.000,C 0.000} C_DIS
WAIT SEC 1.75
RET=EKI_SetBool("oxy","torchState",TRUE)
RET = EKI_Send("oxy","torchState")
LIN {X 181.644,Y -226.065,Z 175.643,A 128.782,B 90.000,C 0.000} C_DIS
LIN {X 183.356,Y -224.679,Z 176.824,A 129.217,B 90.000,C 0.000} C_DIS
LIN {X 184.996,Y -223.330,Z 178.142,A 129.637,B 90.000,C 0.000} C_DIS
LIN {X 186.561,Y -222.024,Z 179.589,A 130.039,B 90.000,C 0.000} C_DIS
LIN {X 188.046,Y -220.769,Z 181.161,A 130.424,B 90.000,C 0.000} C_DIS
LIN {X 189.445,Y -219.569,Z 182.849,A 130.788,B 90.000,C 0.000} C_DIS
LIN {X 190.756,Y -218.431,Z 184.648,A 131.131,B 90.000,C 0.000} C_DIS
LIN {X 191.973,Y -217.362,Z 186.551,A 131.451,B 90.000,C 0.000} C_DIS
LIN {X 193.092,Y -216.368,Z 188.554,A 131.746,B 90.000,C 0.000} C_DIS
LIN {X 194.110,Y -215.456,Z 190.647,A 132.016,B 90.000,C 0.000} C_DIS
LIN {X 194.601,Y -215.012,Z 191.775,A 132.147,B 90.000,C 0.000} C_DIS
LIN {X 193.259,Y -213.530,Z 191.775,A 132.147,B 90.000,C 0.000} C_DIS
WAIT SEC 0.1
RET=EKI_SetBool("oxy","torchState",FALSE)
RET = EKI_Send("oxy","torchState")
LIN {X 181.181,Y -200.184,Z 191.775,A 132.147,B 90.000,C 0.000} C_DIS
LIN {X 185.709,Y -195.990,Z 208.264,A 133.457,B 90.000,C 0.000} C_DIS
LIN {X 198.090,Y -209.056,Z 208.264,A 133.457,B 90.000,C 0.000} C_DIS
LIN {X 199.465,Y -210.508,Z 208.264,A 133.457,B 90.000,C 0.000} C_DIS
WAIT SEC 1.75
RET=EKI_SetBool("oxy","torchState",TRUE)
RET = EKI_Send("oxy","torchState")
LIN {X 200.098,Y -209.907,Z 210.607,A 133.630,B 90.000,C 0.000} C_DIS
LIN {X 200.776,Y -209.258,Z 212.924,A 133.815,B 90.000,C 0.000} C_DIS
LIN {X 201.513,Y -208.549,Z 215.205,A 134.017,B 90.000,C 0.000} C_DIS
LIN {X 202.327,Y -207.759,Z 217.432,A 134.241,B 90.000,C 0.000} C_DIS
LIN {X 203.233,Y -206.873,Z 219.587,A 134.492,B 90.000,C 0.000} C_DIS
LIN {X 204.242,Y -205.877,Z 221.645,A 134.772,B 90.000,C 0.000} C_DIS
LIN {X 205.364,Y -204.757,Z 223.578,A 135.085,B 90.000,C 0.000} C_DIS
LIN {X 205.503,Y -204.618,Z 223.798,A 135.124,B 90.000,C 0.000} C_DIS
LIN {X 204.086,Y -203.206,Z 223.798,A 135.124,B 90.000,C 0.000} C_DIS
WAIT SEC 0.1
RET=EKI_SetBool("oxy","torchState",FALSE)
RET = EKI_Send("oxy","torchState")
LIN {X 191.331,Y -190.506,Z 223.798,A 135.124,B 90.000,C 0.000} C_DIS
LIN {X 179.447,Y -201.739,Z 222.135,A 131.653,B 90.000,C 0.000} C_DIS
LIN {X 191.410,Y -215.188,Z 222.135,A 131.653,B 90.000,C 0.000} C_DIS
LIN {X 192.740,Y -216.683,Z 222.135,A 131.653,B 90.000,C 0.000} C_DIS
WAIT SEC 1.75
RET=EKI_SetBool("oxy","torchState",TRUE)
RET = EKI_Send("oxy","torchState")
LIN {X 193.857,Y -215.684,Z 224.135,A 131.949,B 90.000,C 0.000} C_DIS
LIN {X 194.851,Y -214.786,Z 226.246,A 132.214,B 90.000,C 0.000} C_DIS
LIN {X 195.714,Y -214.000,Z 228.456,A 132.445,B 90.000,C 0.000} C_DIS
LIN {X 196.449,Y -213.325,Z 230.748,A 132.642,B 90.000,C 0.000} C_DIS
LIN {X 197.049,Y -212.771,Z 233.111,A 132.803,B 90.000,C 0.000} C_DIS
LIN {X 197.516,Y -212.338,Z 235.528,A 132.929,B 90.000,C 0.000} C_DIS
LIN {X 197.844,Y -212.032,Z 237.987,A 133.018,B 90.000,C 0.000} C_DIS
LIN {X 198.034,Y -211.855,Z 240.473,A 133.069,B 90.000,C 0.000} C_DIS
LIN {X 198.078,Y -211.814,Z 242.972,A 133.081,B 90.000,C 0.000} C_DIS
LIN {X 198.053,Y -211.838,Z 244.092,A 133.074,B 90.000,C 0.000} C_DIS
LIN {X 196.687,Y -210.377,Z 244.092,A 133.074,B 90.000,C 0.000} C_DIS
WAIT SEC 0.1
RET=EKI_SetBool("oxy","torchState",FALSE)
RET = EKI_Send("oxy","torchState")
LIN {X 184.394,Y -197.228,Z 244.092,A 133.074,B 90.000,C 0.000} C_DIS
LIN {X 202.632,Y -178.438,Z 233.628,A 138.633,B 90.000,C 0.000} C_DIS
LIN {X 216.141,Y -190.334,Z 233.628,A 138.633,B 90.000,C 0.000} C_DIS
LIN {X 217.642,Y -191.656,Z 233.628,A 138.633,B 90.000,C 0.000} C_DIS
WAIT SEC 1.75
RET=EKI_SetBool("oxy","torchState",TRUE)
RET = EKI_Send("oxy","torchState")
LIN {X 219.241,Y -189.824,Z 234.205,A 139.113,B 90.000,C 0.000} C_DIS
LIN {X 220.838,Y -187.963,Z 234.691,A 139.598,B 90.000,C 0.000} C_DIS
LIN {X 222.429,Y -186.078,Z 235.100,A 140.085,B 90.000,C 0.000} C_DIS
LIN {X 224.009,Y -184.173,Z 235.448,A 140.574,B 90.000,C 0.000} C_DIS
LIN {X 225.577,Y -182.249,Z 235.748,A 141.064,B 90.000,C 0.000} C_DIS
LIN {X 227.130,Y -180.309,Z 236.017,A 141.555,B 90.000,C 0.000} C_DIS
LIN {X 228.667,Y -178.354,Z 236.271,A 142.047,B 90.000,C 0.000} C_DIS
LIN {X 230.188,Y -176.387,Z 236.525,A 142.538,B 90.000,C 0.000} C_DIS
LIN {X 230.543,Y -175.926,Z 236.584,A 142.653,B 90.000,C 0.000} C_DIS
LIN {X 228.953,Y -174.713,Z 236.584,A 142.653,B 90.000,C 0.000} C_DIS
WAIT SEC 0.1
RET=EKI_SetBool("oxy","torchState",FALSE)
RET = EKI_Send("oxy","torchState")
LIN {X 214.643,Y -163.793,Z 236.584,A 142.653,B 90.000,C 0.000} C_DIS
LIN {X 210.860,Y -168.636,Z 222.242,A 141.349,B 90.000,C 0.000} C_DIS
LIN {X 224.918,Y -179.878,Z 222.242,A 141.349,B 90.000,C 0.000} C_DIS
LIN {X 226.480,Y -181.127,Z 222.242,A 141.349,B 90.000,C 0.000} C_DIS
WAIT SEC 1.75
RET=EKI_SetBool("oxy","torchState",TRUE)
RET = EKI_Send("oxy","torchState")
LIN {X 225.045,Y -182.907,Z 221.231,A 140.897,B 90.000,C 0.000} C_DIS
LIN {X 223.623,Y -184.642,Z 220.128,A 140.454,B 90.000,C 0.000} C_DIS
LIN {X 222.222,Y -186.326,Z 218.924,A 140.021,B 90.000,C 0.000} C_DIS
LIN {X 220.849,Y -187.951,Z 217.611,A 139.601,B 90.000,C 0.000} C_DIS
LIN {X 219.516,Y -189.506,Z 216.178,A 139.196,B 90.000,C 0.000} C_DIS
LIN {X 218.234,Y -190.981,Z 214.619,A 138.810,B 90.000,C 0.000} C_DIS
LIN {X 217.017,Y -192.364,Z 212.930,A 138.446,B 90.000,C 0.000} C_DIS
LIN {X 216.031,Y -193.470,Z 211.367,A 138.153,B 90.000,C 0.000} C_DIS
LIN {X 214.541,Y -192.136,Z 211.367,A 138.153,B 90.000,C 0.000} C_DIS
WAIT SEC 0.1
RET=EKI_SetBool("oxy","torchState",FALSE)
RET = EKI_Send("oxy","torchState")
LIN {X 201.132,Y -180.127,Z 211.367,A 138.153,B 90.000,C 0.000} C_DIS
LIN {X 212.622,Y -166.409,Z 197.830,A 141.951,B 90.000,C 0.000} C_DIS
LIN {X 226.796,Y -177.503,Z 197.830,A 141.951,B 90.000,C 0.000} C_DIS
LIN {X 228.371,Y -178.736,Z 197.830,A 141.951,B 90.000,C 0.000} C_DIS
WAIT SEC 1.75
RET=EKI_SetBool("oxy","torchState",TRUE)
RET = EKI_Send("oxy","torchState")
LIN {X 227.069,Y -180.387,Z 196.479,A 141.536,B 90.000,C 0.000} C_DIS
LIN {X 225.802,Y -181.971,Z 195.019,A 141.135,B 90.000,C 0.000} C_DIS
LIN {X 224.574,Y -183.484,Z 193.452,A 140.750,B 90.000,C 0.000} C_DIS
LIN {X 223.394,Y -184.919,Z 191.781,A 140.383,B 90.000,C 0.000} C_DIS
LIN {X 222.267,Y -186.272,Z 190.006,A 140.035,B 90.000,C 0.000} C_DIS
LIN {X 221.202,Y -187.536,Z 188.131,A 139.709,B 90.000,C 0.000} C_DIS
LIN {X 220.206,Y -188.704,Z 186.158,A 139.405,B 90.000,C 0.000} C_DIS
LIN {X 219.289,Y -189.769,Z 184.091,A 139.128,B 90.000,C 0.000} C_DIS
LIN {X 218.459,Y -190.724,Z 181.935,A 138.878,B 90.000,C 0.000} C_DIS
LIN {X 217.888,Y -191.376,Z 180.235,A 138.706,B 90.000,C 0.000} C_DIS
LIN {X 216.385,Y -190.056,Z 180.235,A 138.706,B 90.000,C 0.000} C_DIS
WAIT SEC 0.1
RET=EKI_SetBool("oxy","torchState",FALSE)
RET = EKI_Send("oxy","torchState")
LIN {X 202.861,Y -178.178,Z 180.235,A 138.706,B 90.000,C 0.000} C_DIS
LIN {X 194.646,Y -187.118,Z 189.743,A 136.130,B 90.000,C 0.000} C_DIS
LIN {X 207.622,Y -199.592,Z 189.743,A 136.130,B 90.000,C 0.000} C_DIS
LIN {X 209.064,Y -200.979,Z 189.743,A 136.130,B 90.000,C 0.000} C_DIS
WAIT SEC 1.75
RET=EKI_SetBool("oxy","torchState",TRUE)
RET = EKI_Send("oxy","torchState")
LIN {X 208.624,Y -201.435,Z 187.325,A 136.004,B 90.000,C 0.000} C_DIS
LIN {X 208.197,Y -201.876,Z 184.902,A 135.883,B 90.000,C 0.000} C_DIS
LIN {X 207.772,Y -202.313,Z 182.477,A 135.763,B 90.000,C 0.000} C_DIS
LIN {X 207.342,Y -202.754,Z 180.055,A 135.641,B 90.000,C 0.000} C_DIS
LIN {X 206.892,Y -203.213,Z 177.639,A 135.514,B 90.000,C 0.000} C_DIS
LIN {X 206.412,Y -203.701,Z 175.235,A 135.379,B 90.000,C 0.000} C_DIS
LIN {X 205.890,Y -204.228,Z 172.848,A 135.232,B 90.000,C 0.000} C_DIS
LIN {X 205.316,Y -204.806,Z 170.485,A 135.071,B 90.000,C 0.000} C_DIS
LIN {X 204.678,Y -205.444,Z 168.153,A 134.893,B 90.000,C 0.000} C_DIS
LIN {X 204.218,Y -205.901,Z 166.637,A 134.765,B 90.000,C 0.000} C_DIS
LIN {X 202.809,Y -204.481,Z 166.637,A 134.765,B 90.000,C 0.000} C_DIS
WAIT SEC 0.1
RET=EKI_SetBool("oxy","torchState",FALSE)
RET = EKI_Send("oxy","torchState")
LIN {X 190.134,Y -191.701,Z 166.637,A 134.765,B 90.000,C 0.000} C_DIS
LIN {X 199.026,Y -182.452,Z 158.114,A 137.488,B 90.000,C 0.000} C_DIS
LIN {X 212.295,Y -194.615,Z 158.114,A 137.488,B 90.000,C 0.000} C_DIS
LIN {X 213.769,Y -195.967,Z 158.114,A 137.488,B 90.000,C 0.000} C_DIS
WAIT SEC 1.75
RET=EKI_SetBool("oxy","torchState",TRUE)
RET = EKI_Send("oxy","torchState")
LIN {X 213.332,Y -196.442,Z 155.700,A 137.360,B 90.000,C 0.000} C_DIS
LIN {X 212.848,Y -196.966,Z 153.304,A 137.219,B 90.000,C 0.000} C_DIS
LIN {X 212.312,Y -197.544,Z 150.932,A 137.064,B 90.000,C 0.000} C_DIS
LIN {X 211.722,Y -198.176,Z 148.586,A 136.893,B 90.000,C 0.000} C_DIS
LIN {X 211.076,Y -198.864,Z 146.272,A 136.706,B 90.000,C 0.000} C_DIS
LIN {X 210.368,Y -199.613,Z 143.994,A 136.503,B 90.000,C 0.000} C_DIS
LIN {X 209.598,Y -200.421,Z 141.757,A 136.282,B 90.000,C 0.000} C_DIS
LIN {X 208.761,Y -201.293,Z 139.569,A 136.043,B 90.000,C 0.000} C_DIS
LIN {X 208.219,Y -201.853,Z 138.260,A 135.889,B 90.000,C 0.000} C_DIS
LIN {X 206.783,Y -200.461,Z 138.260,A 135.889,B 90.000,C 0.000} C_DIS
WAIT SEC 0.1
RET=EKI_SetBool("oxy","torchState",FALSE)
RET = EKI_Send("oxy","torchState")
LIN {X 193.859,Y -187.932,Z 138.260,A 135.889,B 90.000,C 0.000} C_DIS
LIN {X 229.894,Y -141.593,Z 174.838,A 148.371,B 90.000,C 0.000} C_DIS
LIN {X 245.220,Y -151.033,Z 174.838,A 148.371,B 90.000,C 0.000} C_DIS
LIN {X 246.923,Y -152.082,Z 174.838,A 148.371,B 90.000,C 0.000} C_DIS
WAIT SEC 1.75
RET=EKI_SetBool("oxy","torchState",TRUE)
RET = EKI_Send("oxy","torchState")
LIN {X 248.223,Y -149.951,Z 174.701,A 148.864,B 90.000,C 0.000} C_DIS
LIN {X 249.489,Y -147.835,Z 174.291,A 149.351,B 90.000,C 0.000} C_DIS
LIN {X 250.707,Y -145.760,Z 173.613,A 149.826,B 90.000,C 0.000} C_DIS
LIN {X 251.864,Y -143.751,Z 172.679,A 150.285,B 90.000,C 0.000} C_DIS
LIN {X 252.949,Y -141.833,Z 171.498,A 150.720,B 90.000,C 0.000} C_DIS
LIN {X 253.952,Y -140.029,Z 170.088,A 151.128,B 90.000,C 0.000} C_DIS
LIN {X 254.043,Y -139.864,Z 169.944,A 151.165,B 90.000,C 0.000} C_DIS
LIN {X 252.829,Y -142.048,Z 169.881,A 150.671,B 90.000,C 0.000} C_DIS
LIN {X 251.613,Y -144.190,Z 169.455,A 150.185,B 90.000,C 0.000} C_DIS
LIN {X 250.424,Y -146.246,Z 168.674,A 149.715,B 90.000,C 0.000} C_DIS
LIN {X 249.288,Y -148.173,Z 167.560,A 149.273,B 90.000,C 0.000} C_DIS
LIN {X 248.230,Y -149.939,Z 166.141,A 148.867,B 90.000,C 0.000} C_DIS
LIN {X 247.273,Y -151.512,Z 164.451,A 148.503,B 90.000,C 0.000} C_DIS
LIN {X 246.434,Y -152.874,Z 162.530,A 148.187,B 90.000,C 0.000} C_DIS
LIN {X 245.730,Y -154.002,Z 160.413,A 147.924,B 90.000,C 0.000} C_DIS
LIN {X 245.175,Y -154.885,Z 158.141,A 147.718,B 90.000,C 0.000} C_DIS
LIN {X 244.778,Y -155.510,Z 155.754,A 147.572,B 90.000,C 0.000} C_DIS
LIN {X 244.547,Y -155.874,Z 153.292,A 147.487,B 90.000,C 0.000} C_DIS
LIN {X 244.484,Y -155.973,Z 150.795,A 147.463,B 90.000,C 0.000} C_DIS
LIN {X 244.588,Y -155.810,Z 148.302,A 147.502,B 90.000,C 0.000} C_DIS
LIN {X 244.859,Y -155.384,Z 145.854,A 147.601,B 90.000,C 0.000} C_DIS
LIN {X 245.295,Y -154.694,Z 143.492,A 147.763,B 90.000,C 0.000} C_DIS
LIN {X 245.887,Y -153.752,Z 141.253,A 147.983,B 90.000,C 0.000} C_DIS
LIN {X 246.625,Y -152.565,Z 139.181,A 148.259,B 90.000,C 0.000} C_DIS
LIN {X 247.494,Y -151.151,Z 137.312,A 148.587,B 90.000,C 0.000} C_DIS
LIN {X 248.478,Y -149.529,Z 135.684,A 148.961,B 90.000,C 0.000} C_DIS
LIN {X 249.557,Y -147.721,Z 134.336,A 149.377,B 90.000,C 0.000} C_DIS
LIN {X 250.708,Y -145.759,Z 133.300,A 149.827,B 90.000,C 0.000} C_DIS
LIN {X 251.906,Y -143.678,Z 132.603,A 150.301,B 90.000,C 0.000} C_DIS
LIN {X 253.124,Y -141.522,Z 132.264,A 150.790,B 90.000,C 0.000} C_DIS
LIN {X 254.125,Y -139.715,Z 132.259,A 151.198,B 90.000,C 0.000} C_DIS
LIN {X 254.010,Y -139.924,Z 132.072,A 151.151,B 90.000,C 0.000} C_DIS
LIN {X 253.012,Y -141.721,Z 130.648,A 150.745,B 90.000,C 0.000} C_DIS
LIN {X 251.932,Y -143.633,Z 129.454,A 150.311,B 90.000,C 0.000} C_DIS
LIN {X 250.778,Y -145.637,Z 128.505,A 149.855,B 90.000,C 0.000} C_DIS
LIN {X 249.563,Y -147.709,Z 127.813,A 149.380,B 90.000,C 0.000} C_DIS
LIN {X 248.300,Y -149.824,Z 127.387,A 148.893,B 90.000,C 0.000} C_DIS
LIN {X 247.002,Y -151.954,Z 127.233,A 148.400,B 90.000,C 0.000} C_DIS
LIN {X 245.684,Y -154.075,Z 127.354,A 147.907,B 90.000,C 0.000} C_DIS
LIN {X 244.364,Y -156.161,Z 127.747,A 147.419,B 90.000,C 0.000} C_DIS
LIN {X 243.057,Y -158.187,Z 128.408,A 146.943,B 90.000,C 0.000} C_DIS
LIN {X 241.781,Y -160.130,Z 129.327,A 146.484,B 90.000,C 0.000} C_DIS
LIN {X 240.554,Y -161.969,Z 130.493,A 146.047,B 90.000,C 0.000} C_DIS
LIN {X 239.390,Y -163.684,Z 131.891,A 145.637,B 90.000,C 0.000} C_DIS
LIN {X 238.306,Y -165.258,Z 133.502,A 145.260,B 90.000,C 0.000} C_DIS
LIN {X 237.317,Y -166.676,Z 135.307,A 144.918,B 90.000,C 0.000} C_DIS
LIN {X 236.434,Y -167.925,Z 137.285,A 144.616,B 90.000,C 0.000} C_DIS
LIN {X 235.672,Y -168.994,Z 139.412,A 144.357,B 90.000,C 0.000} C_DIS
LIN {X 235.038,Y -169.874,Z 141.664,A 144.142,B 90.000,C 0.000} C_DIS
LIN {X 234.542,Y -170.558,Z 144.017,A 143.975,B 90.000,C 0.000} C_DIS
LIN {X 234.190,Y -171.041,Z 146.444,A 143.857,B 90.000,C 0.000} C_DIS
LIN {X 233.986,Y -171.320,Z 148.920,A 143.789,B 90.000,C 0.000} C_DIS
LIN {X 233.934,Y -171.392,Z 151.418,A 143.772,B 90.000,C 0.000} C_DIS
LIN {X 234.033,Y -171.256,Z 153.912,A 143.805,B 90.000,C 0.000} C_DIS
LIN {X 234.282,Y -170.915,Z 156.375,A 143.888,B 90.000,C 0.000} C_DIS
LIN {X 234.679,Y -170.370,Z 158.783,A 144.021,B 90.000,C 0.000} C_DIS
LIN {X 235.218,Y -169.625,Z 161.107,A 144.203,B 90.000,C 0.000} C_DIS
LIN {X 235.892,Y -168.686,Z 163.324,A 144.431,B 90.000,C 0.000} C_DIS
LIN {X 236.692,Y -167.561,Z 165.407,A 144.704,B 90.000,C 0.000} C_DIS
LIN {X 237.608,Y -166.260,Z 167.335,A 145.019,B 90.000,C 0.000} C_DIS
LIN {X 238.628,Y -164.792,Z 169.082,A 145.372,B 90.000,C 0.000} C_DIS
LIN {X 239.738,Y -163.173,Z 170.630,A 145.760,B 90.000,C 0.000} C_DIS
LIN {X 240.923,Y -161.418,Z 171.959,A 146.178,B 90.000,C 0.000} C_DIS
LIN {X 242.168,Y -159.546,Z 173.051,A 146.622,B 90.000,C 0.000} C_DIS
LIN {X 243.455,Y -157.575,Z 173.892,A 147.087,B 90.000,C 0.000} C_DIS
LIN {X 244.767,Y -155.528,Z 174.472,A 147.568,B 90.000,C 0.000} C_DIS
LIN {X 246.089,Y -153.429,Z 174.781,A 148.058,B 90.000,C 0.000} C_DIS
LIN {X 246.924,Y -152.081,Z 174.838,A 148.371,B 90.000,C 0.000} C_DIS
LIN {X 245.221,Y -151.032,Z 174.838,A 148.371,B 90.000,C 0.000} C_DIS
WAIT SEC 0.1
RET=EKI_SetBool("oxy","torchState",FALSE)
RET = EKI_Send("oxy","torchState")
LIN {X 229.894,Y -141.593,Z 174.838,A 148.371,B 90.000,C 0.000} C_DIS
LIN {X 165.071,Y -213.662,Z 210.677,A 127.689,B 90.000,C 0.000} C_DIS
LIN {X 176.076,Y -227.906,Z 210.677,A 127.689,B 90.000,C 0.000} C_DIS
LIN {X 177.299,Y -229.489,Z 210.677,A 127.689,B 90.000,C 0.000} C_DIS
WAIT SEC 1.75
RET=EKI_SetBool("oxy","torchState",TRUE)
RET = EKI_Send("oxy","torchState")
LIN {X 175.326,Y -230.999,Z 210.403,A 127.198,B 90.000,C 0.000} C_DIS
LIN {X 173.329,Y -232.501,Z 210.341,A 126.704,B 90.000,C 0.000} C_DIS
LIN {X 171.324,Y -233.983,Z 210.515,A 126.212,B 90.000,C 0.000} C_DIS
LIN {X 169.331,Y -235.430,Z 210.945,A 125.725,B 90.000,C 0.000} C_DIS
LIN {X 167.372,Y -236.826,Z 211.625,A 125.250,B 90.000,C 0.000} C_DIS
LIN {X 165.469,Y -238.160,Z 212.545,A 124.791,B 90.000,C 0.000} C_DIS
LIN {X 163.640,Y -239.420,Z 213.693,A 124.352,B 90.000,C 0.000} C_DIS
LIN {X 161.907,Y -240.595,Z 215.058,A 123.938,B 90.000,C 0.000} C_DIS
LIN {X 160.291,Y -241.675,Z 216.629,A 123.554,B 90.000,C 0.000} C_DIS
LIN {X 159.332,Y -242.308,Z 217.729,A 123.327,B 90.000,C 0.000} C_DIS
LIN {X 158.233,Y -240.637,Z 217.729,A 123.327,B 90.000,C 0.000} C_DIS
WAIT SEC 0.1
RET=EKI_SetBool("oxy","torchState",FALSE)
RET = EKI_Send("oxy","torchState")
LIN {X 148.344,Y -225.597,Z 217.729,A 123.327,B 90.000,C 0.000} C_DIS
LIN {X 269.043,Y -22.716,Z 237.590,A 175.174,B 90.000,C 0.000} C_DIS
LIN {X 286.979,Y -24.230,Z 237.590,A 175.174,B 90.000,C 0.000} C_DIS
LIN {X 288.972,Y -24.399,Z 237.590,A 175.174,B 90.000,C 0.000} C_DIS
WAIT SEC 1.75
RET=EKI_SetBool("oxy","torchState",TRUE)
RET = EKI_Send("oxy","torchState")
LIN {X 289.170,Y -21.920,Z 237.848,A 175.665,B 90.000,C 0.000} C_DIS
LIN {X 289.345,Y -19.473,Z 238.328,A 176.150,B 90.000,C 0.000} C_DIS
LIN {X 289.497,Y -17.078,Z 239.026,A 176.624,B 90.000,C 0.000} C_DIS
LIN {X 289.624,Y -14.753,Z 239.936,A 177.084,B 90.000,C 0.000} C_DIS
LIN {X 289.730,Y -12.517,Z 241.048,A 177.526,B 90.000,C 0.000} C_DIS
LIN {X 289.814,Y -10.388,Z 242.355,A 177.947,B 90.000,C 0.000} C_DIS
LIN {X 289.865,Y -8.852,Z 243.477,A 178.251,B 90.000,C 0.000} C_DIS
LIN {X 287.866,Y -8.791,Z 243.477,A 178.251,B 90.000,C 0.000} C_DIS
WAIT SEC 0.1
RET=EKI_SetBool("oxy","torchState",FALSE)
RET = EKI_Send("oxy","torchState")
LIN {X 269.874,Y -8.241,Z 243.477,A 178.251,B 90.000,C 0.000} C_DIS
LIN {X 253.612,Y 92.635,Z 169.381,A -159.935,B 90.000,C 0.000} C_DIS
LIN {X 270.519,Y 98.810,Z 169.381,A -159.935,B 90.000,C 0.000} C_DIS
LIN {X 272.398,Y 99.496,Z 169.381,A -159.935,B 90.000,C 0.000} C_DIS
WAIT SEC 1.75
RET=EKI_SetBool("oxy","torchState",TRUE)
RET = EKI_Send("oxy","torchState")
LIN {X 271.581,Y 101.698,Z 170.237,A -159.471,B 90.000,C 0.000} C_DIS
LIN {X 270.747,Y 103.891,Z 171.101,A -159.007,B 90.000,C 0.000} C_DIS
LIN {X 269.898,Y 106.076,Z 171.968,A -158.544,B 90.000,C 0.000} C_DIS
LIN {X 269.029,Y 108.252,Z 172.840,A -158.081,B 90.000,C 0.000} C_DIS
LIN {X 268.150,Y 110.424,Z 173.711,A -157.618,B 90.000,C 0.000} C_DIS
LIN {X 267.248,Y 112.587,Z 174.581,A -157.155,B 90.000,C 0.000} C_DIS
LIN {X 266.332,Y 114.744,Z 175.449,A -156.692,B 90.000,C 0.000} C_DIS
LIN {X 265.396,Y 116.896,Z 176.311,A -156.228,B 90.000,C 0.000} C_DIS
LIN {X 264.440,Y 119.042,Z 177.164,A -155.764,B 90.000,C 0.000} C_DIS
LIN {X 263.465,Y 121.184,Z 178.007,A -155.299,B 90.000,C 0.000} C_DIS
LIN {X 262.472,Y 123.322,Z 178.838,A -154.834,B 90.000,C 0.000} C_DIS
LIN {X 261.458,Y 125.457,Z 179.653,A -154.367,B 90.000,C 0.000} C_DIS
LIN {X 260.425,Y 127.588,Z 180.451,A -153.899,B 90.000,C 0.000} C_DIS
LIN {X 259.370,Y 129.717,Z 181.229,A -153.429,B 90.000,C 0.000} C_DIS
LIN {X 258.295,Y 131.843,Z 181.986,A -152.959,B 90.000,C 0.000} C_DIS
LIN {X 257.200,Y 133.968,Z 182.718,A -152.486,B 90.000,C 0.000} C_DIS
LIN {X 256.085,Y 136.090,Z 183.426,A -152.013,B 90.000,C 0.000} C_DIS
LIN {X 254.946,Y 138.210,Z 184.101,A -151.537,B 90.000,C 0.000} C_DIS
LIN {X 253.786,Y 140.329,Z 184.746,A -151.060,B 90.000,C 0.000} C_DIS
LIN {X 252.604,Y 142.445,Z 185.357,A -150.581,B 90.000,C 0.000} C_DIS
LIN {X 251.401,Y 144.559,Z 185.932,A -150.101,B 90.000,C 0.000} C_DIS
LIN {X 251.176,Y 144.951,Z 186.036,A -150.011,B 90.000,C 0.000} C_DIS
LIN {X 249.443,Y 143.951,Z 186.036,A -150.011,B 90.000,C 0.000} C_DIS
WAIT SEC 0.1
RET=EKI_SetBool("oxy","torchState",FALSE)
RET = EKI_Send("oxy","torchState")
LIN {X 233.853,Y 134.954,Z 186.036,A -150.011,B 90.000,C 0.000} C_DIS
LIN {X 244.014,Y 115.573,Z 138.293,A -154.656,B 90.000,C 0.000} C_DIS
LIN {X 260.282,Y 123.278,Z 138.293,A -154.656,B 90.000,C 0.000} C_DIS
LIN {X 262.089,Y 124.134,Z 138.293,A -154.656,B 90.000,C 0.000} C_DIS
WAIT SEC 1.75
RET=EKI_SetBool("oxy","torchState",TRUE)
RET = EKI_Send("oxy","torchState")
LIN {X 263.104,Y 121.966,Z 137.574,A -155.129,B 90.000,C 0.000} C_DIS
LIN {X 264.102,Y 119.787,Z 136.861,A -155.603,B 90.000,C 0.000} C_DIS
LIN {X 265.080,Y 117.597,Z 136.156,A -156.076,B 90.000,C 0.000} C_DIS
LIN {X 266.048,Y 115.403,Z 135.453,A -156.550,B 90.000,C 0.000} C_DIS
LIN {X 266.993,Y 113.196,Z 134.755,A -157.025,B 90.000,C 0.000} C_DIS
LIN {X 267.917,Y 110.980,Z 134.061,A -157.499,B 90.000,C 0.000} C_DIS
LIN {X 268.833,Y 108.760,Z 133.368,A -157.974,B 90.000,C 0.000} C_DIS
LIN {X 269.718,Y 106.526,Z 132.677,A -158.448,B 90.000,C 0.000} C_DIS
LIN {X 270.596,Y 104.290,Z 131.985,A -158.923,B 90.000,C 0.000} C_DIS
LIN {X 271.452,Y 102.046,Z 131.292,A -159.397,B 90.000,C 0.000} C_DIS
LIN {X 272.287,Y 99.794,Z 130.600,A -159.872,B 90.000,C 0.000} C_DIS
LIN {X 273.097,Y 97.535,Z 129.902,A -160.346,B 90.000,C 0.000} C_DIS
LIN {X 273.903,Y 95.274,Z 129.204,A -160.820,B 90.000,C 0.000} C_DIS
LIN {X 274.676,Y 93.004,Z 128.499,A -161.294,B 90.000,C 0.000} C_DIS
LIN {X 275.437,Y 90.731,Z 127.789,A -161.768,B 90.000,C 0.000} C_DIS
LIN {X 276.180,Y 88.454,Z 127.075,A -162.241,B 90.000,C 0.000} C_DIS
LIN {X 276.898,Y 86.171,Z 126.350,A -162.714,B 90.000,C 0.000} C_DIS
LIN {X 277.166,Y 85.317,Z 126.079,A -162.891,B 90.000,C 0.000} C_DIS
LIN {X 275.255,Y 84.729,Z 126.079,A -162.891,B 90.000,C 0.000} C_DIS
WAIT SEC 0.1
RET=EKI_SetBool("oxy","torchState",FALSE)
RET = EKI_Send("oxy","torchState")
LIN {X 258.051,Y 79.433,Z 126.079,A -162.891,B 90.000,C 0.000} C_DIS
LIN {X 216.536,Y 161.282,Z 91.013,A -143.320,B 90.000,C 0.000} C_DIS
LIN {X 230.972,Y 172.035,Z 91.013,A -143.320,B 90.000,C 0.000} C_DIS
LIN {X 232.576,Y 173.229,Z 91.013,A -143.320,B 90.000,C 0.000} C_DIS
WAIT SEC 1.75
RET=EKI_SetBool("oxy","torchState",TRUE)
RET = EKI_Send("oxy","torchState")
LIN {X 231.162,Y 175.111,Z 91.855,A -142.855,B 90.000,C 0.000} C_DIS
LIN {X 229.744,Y 176.967,Z 92.745,A -142.394,B 90.000,C 0.000} C_DIS
LIN {X 228.318,Y 178.804,Z 93.661,A -141.934,B 90.000,C 0.000} C_DIS
LIN {X 226.877,Y 180.625,Z 94.587,A -141.475,B 90.000,C 0.000} C_DIS
LIN {X 225.423,Y 182.440,Z 95.505,A -141.016,B 90.000,C 0.000} C_DIS
LIN {X 223.947,Y 184.249,Z 96.395,A -140.555,B 90.000,C 0.000} C_DIS
LIN {X 222.444,Y 186.060,Z 97.238,A -140.090,B 90.000,C 0.000} C_DIS
LIN {X 221.117,Y 187.636,Z 97.922,A -139.683,B 90.000,C 0.000} C_DIS
LIN {X 219.592,Y 186.342,Z 97.922,A -139.683,B 90.000,C 0.000} C_DIS
WAIT SEC 0.1
RET=EKI_SetBool("oxy","torchState",FALSE)
RET = EKI_Send("oxy","torchState")
LIN {X 205.868,Y 174.695,Z 97.922,A -139.683,B 90.000,C 0.000} C_DIS
LIN {X 193.748,Y 188.048,Z 99.649,A -135.855,B 90.000,C 0.000} C_DIS
LIN {X 206.664,Y 200.584,Z 99.649,A -135.855,B 90.000,C 0.000} C_DIS
LIN {X 208.099,Y 201.977,Z 99.649,A -135.855,B 90.000,C 0.000} C_DIS
WAIT SEC 1.75
RET=EKI_SetBool("oxy","torchState",TRUE)
RET = EKI_Send("oxy","torchState")
LIN {X 206.408,Y 203.704,Z 99.012,A -135.378,B 90.000,C 0.000} C_DIS
LIN {X 204.752,Y 205.369,Z 98.156,A -134.914,B 90.000,C 0.000} C_DIS
LIN {X 203.140,Y 206.964,Z 97.104,A -134.466,B 90.000,C 0.000} C_DIS
LIN {X 201.581,Y 208.483,Z 95.875,A -134.036,B 90.000,C 0.000} C_DIS
LIN {X 200.077,Y 209.926,Z 94.495,A -133.624,B 90.000,C 0.000} C_DIS
LIN {X 198.633,Y 211.294,Z 92.981,A -133.231,B 90.000,C 0.000} C_DIS
LIN {X 197.247,Y 212.588,Z 91.353,A -132.856,B 90.000,C 0.000} C_DIS
LIN {X 195.919,Y 213.813,Z 89.625,A -132.499,B 90.000,C 0.000} C_DIS
LIN {X 194.648,Y 214.970,Z 87.810,A -132.160,B 90.000,C 0.000} C_DIS
LIN {X 193.667,Y 215.854,Z 86.302,A -131.899,B 90.000,C 0.000} C_DIS
LIN {X 192.332,Y 214.365,Z 86.302,A -131.899,B 90.000,C 0.000} C_DIS
WAIT SEC 0.1
RET=EKI_SetBool("oxy","torchState",FALSE)
RET = EKI_Send("oxy","torchState")
LIN {X 180.311,Y 200.967,Z 86.302,A -131.899,B 90.000,C 0.000} C_DIS
LIN {X 169.598,Y 210.087,Z 69.815,A -128.913,B 90.000,C 0.000} C_DIS
LIN {X 180.904,Y 224.093,Z 69.815,A -128.913,B 90.000,C 0.000} C_DIS
LIN {X 182.160,Y 225.649,Z 69.815,A -128.913,B 90.000,C 0.000} C_DIS
WAIT SEC 1.75
RET=EKI_SetBool("oxy","torchState",TRUE)
RET = EKI_Send("oxy","torchState")
LIN {X 180.472,Y 227.002,Z 68.562,A -128.486,B 90.000,C 0.000} C_DIS
LIN {X 178.691,Y 228.407,Z 67.513,A -128.037,B 90.000,C 0.000} C_DIS
LIN {X 176.839,Y 229.843,Z 66.642,A -127.574,B 90.000,C 0.000} C_DIS
LIN {X 174.935,Y 231.296,Z 65.926,A -127.101,B 90.000,C 0.000} C_DIS
LIN {X 172.992,Y 232.752,Z 65.334,A -126.621,B 90.000,C 0.000} C_DIS
LIN {X 171.020,Y 234.205,Z 64.835,A -126.137,B 90.000,C 0.000} C_DIS
LIN {X 169.026,Y 235.649,Z 64.400,A -125.651,B 90.000,C 0.000} C_DIS
LIN {X 167.014,Y 237.079,Z 64.007,A -125.163,B 90.000,C 0.000} C_DIS
LIN {X 164.984,Y 238.495,Z 63.661,A -124.674,B 90.000,C 0.000} C_DIS
LIN {X 162.935,Y 239.900,Z 63.384,A -124.183,B 90.000,C 0.000} C_DIS
LIN {X 160.866,Y 241.292,Z 63.201,A -123.691,B 90.000,C 0.000} C_DIS
LIN {X 158.781,Y 242.669,Z 63.137,A -123.197,B 90.000,C 0.000} C_DIS
LIN {X 158.329,Y 242.965,Z 63.141,A -123.090,B 90.000,C 0.000} C_DIS
LIN {X 157.237,Y 241.289,Z 63.141,A -123.090,B 90.000,C 0.000} C_DIS
WAIT SEC 0.1
RET=EKI_SetBool("oxy","torchState",FALSE)
RET = EKI_Send("oxy","torchState")
LIN {X 147.410,Y 226.209,Z 63.141,A -123.090,B 90.000,C 0.000} C_DIS
LIN {X 154.069,Y 221.727,Z 43.704,A -124.794,B 90.000,C 0.000} C_DIS
LIN {X 164.340,Y 236.508,Z 43.704,A -124.794,B 90.000,C 0.000} C_DIS
LIN {X 165.482,Y 238.151,Z 43.704,A -124.794,B 90.000,C 0.000} C_DIS
WAIT SEC 1.75
RET=EKI_SetBool("oxy","torchState",TRUE)
RET = EKI_Send("oxy","torchState")
LIN {X 167.476,Y 236.752,Z 44.265,A -125.275,B 90.000,C 0.000} C_DIS
LIN {X 169.446,Y 235.346,Z 44.888,A -125.753,B 90.000,C 0.000} C_DIS
LIN {X 171.392,Y 233.932,Z 45.568,A -126.229,B 90.000,C 0.000} C_DIS
LIN {X 173.316,Y 232.511,Z 46.297,A -126.701,B 90.000,C 0.000} C_DIS
LIN {X 175.216,Y 231.082,Z 47.069,A -127.171,B 90.000,C 0.000} C_DIS
LIN {X 177.095,Y 229.645,Z 47.878,A -127.638,B 90.000,C 0.000} C_DIS
LIN {X 178.954,Y 228.200,Z 48.715,A -128.103,B 90.000,C 0.000} C_DIS
LIN {X 180.795,Y 226.745,Z 49.577,A -128.567,B 90.000,C 0.000} C_DIS
LIN {X 182.619,Y 225.278,Z 50.456,A -129.029,B 90.000,C 0.000} C_DIS
LIN {X 184.427,Y 223.799,Z 51.345,A -129.491,B 90.000,C 0.000} C_DIS
LIN {X 186.222,Y 222.307,Z 52.239,A -129.952,B 90.000,C 0.000} C_DIS
LIN {X 188.006,Y 220.799,Z 53.130,A -130.414,B 90.000,C 0.000} C_DIS
LIN {X 189.780,Y 219.277,Z 54.014,A -130.876,B 90.000,C 0.000} C_DIS
LIN {X 191.547,Y 217.737,Z 54.884,A -131.339,B 90.000,C 0.000} C_DIS
LIN {X 193.306,Y 216.177,Z 55.733,A -131.803,B 90.000,C 0.000} C_DIS
LIN {X 195.059,Y 214.596,Z 56.554,A -132.270,B 90.000,C 0.000} C_DIS
LIN {X 196.808,Y 212.993,Z 57.343,A -132.738,B 90.000,C 0.000} C_DIS
LIN {X 198.553,Y 211.368,Z 58.092,A -133.209,B 90.000,C 0.000} C_DIS
LIN {X 200.295,Y 209.718,Z 58.792,A -133.684,B 90.000,C 0.000} C_DIS
LIN {X 201.411,Y 208.647,Z 59.216,A -133.989,B 90.000,C 0.000} C_DIS
LIN {X 200.022,Y 207.208,Z 59.216,A -133.989,B 90.000,C 0.000} C_DIS
WAIT SEC 0.1
RET=EKI_SetBool("oxy","torchState",FALSE)
RET = EKI_Send("oxy","torchState")
LIN {X 187.521,Y 194.257,Z 59.216,A -133.989,B 90.000,C 0.000} C_DIS
LIN {X 113.545,Y 244.964,Z 45.261,A -114.868,B 90.000,C 0.000} C_DIS
LIN {X 121.115,Y 261.295,Z 45.261,A -114.868,B 90.000,C 0.000} C_DIS
LIN {X 121.956,Y 263.110,Z 45.261,A -114.868,B 90.000,C 0.000} C_DIS
WAIT SEC 1.75
RET=EKI_SetBool("oxy","torchState",TRUE)
RET = EKI_Send("oxy","torchState")
LIN {X 119.743,Y 264.122,Z 45.834,A -114.388,B 90.000,C 0.000} C_DIS
LIN {X 117.527,Y 265.115,Z 46.427,A -113.908,B 90.000,C 0.000} C_DIS
LIN {X 115.304,Y 266.089,Z 47.027,A -113.429,B 90.000,C 0.000} C_DIS
LIN {X 113.074,Y 267.047,Z 47.624,A -112.949,B 90.000,C 0.000} C_DIS
LIN {X 110.831,Y 267.986,Z 48.204,A -112.469,B 90.000,C 0.000} C_DIS
LIN {X 108.574,Y 268.908,Z 48.754,A -111.987,B 90.000,C 0.000} C_DIS
LIN {X 106.300,Y 269.815,Z 49.259,A -111.503,B 90.000,C 0.000} C_DIS
